// TIA Portal project "FactoryIO_Template_S7-1200_V15 (1)_V16" (V16)
// Vorlageprojekt für das Buch mit Zielsystem S7-1200

(* hardware
DEVICE "S7-1200-Station_1"  S7-1200 Station
   slot 0: "Baugruppenträger_0"  Rack  V1.0
   slot 1: "PLC_1"  CPU 1211C DC/DC/DC  6ES7 211-1AE40-0XB0  V4.1
*)

// ===== PLC "PLC_1"  CPU 1211C DC/DC/DC =====

VAR_GLOBAL   // PLC tag table "Standard-Variablentabelle"
   "visionsensor_1" AT %I0.4 : Bool;
   "pusher_1+" AT %Q0.4 : Bool;
   "pusher_1-" AT %Q0.5 : Bool;
   "pusher_2+" AT %Q0.6 : Bool;
   "visionsensor_2" AT %I0.5 : Bool;
   "visionsensor_3" AT %I0.6 : Bool;
   "visionsensor_4" AT %I0.7 : Bool;
   "pusher_2-" AT %Q0.7 : Bool;
   "pusher_3+" AT %Q1.0 : Bool;
   "pusher_3-" AT %Q1.1 : Bool;
   "pusher_4+" AT %Q1.2 : Bool;
   "pusher_4-" AT %Q1.3 : Bool;
   "Tag_1" AT %I2.5 : Bool;
   "green_moving_x" AT %I2.6 : Bool;
   "Tag_3" AT %MD10 : Time;
   "lids_sensor_bule_1" AT %I1.1 : Bool;
   "blue_lids_clamp" AT %Q2.7 : Bool;
   "blue_move_z" AT %Q2.5 : Bool;
   "blue_grab" AT %Q2.6 : Bool;
   "base_sensor_bule_1" AT %I1.2 : Bool;
   "blue_base_clamp" AT %Q3.0 : Bool;
   "bule_dectected" AT %I2.2 : Bool;
   "Tag_5" AT %MD11 : Time;
   "blue_moving_x" AT %I2.0 : Bool;
   "blue_move_x" AT %Q2.4 : Bool;
   "Tag_4" AT %MD9 : Time;
   "Tag_6" AT %MD12 : Time;
   "Tag_7" AT %MD13 : Time;
   "Start_btn" AT %I0.0 : Bool;
   "sys_on" AT %M99.0 : Bool;
   "stop_btn" AT %I0.2 : Bool;
   "emergency_stop" AT %I0.3 : Bool;
   "Tag_9" AT %M1.1 : Bool;
   "Tag_10" AT %M1.5 : Bool;
   "Tag_11" AT %M5.0 : Bool;
   "Tag_12" AT %M5.1 : Bool;
   "Tag_13" AT %M5.3 : Bool;
   "blue_base_clamped" AT %I2.4 : Bool;
   "Tag_15" AT %M6.1 : Bool;
   "blue_raise_base" AT %Q3.1 : Bool;
   "Tag_16" AT %M6.0 : Bool;
   "Tag_17" AT %M5.6 : Bool;
   "blue_base_sensor_2" AT %I1.3 : Bool;
   "Tag_18" AT %M2.6 : Bool;
   "start_light" AT %Q0.0 : Bool;
   "reset_btn" AT %I0.1 : Bool;
   "reset_light" AT %Q0.1 : Bool;
   "stop_light" AT %Q0.2 : Bool;
   "blue_lids_clamped" AT %I2.3 : Bool;
   "blue_moving_z" AT %I2.1 : Bool;
   "Tag_8" AT %M5.4 : Bool;
   "blue_lids_conveyor" AT %Q2.0 : Bool;
   "blue_base_conveyor" AT %Q2.1 : Bool;
   "Tag_19" AT %M0.7 : Bool;
   "Tag_20" AT %M0.5 : Bool;
   "Tag_21" AT %M10.1 : Bool;
   "Tag_22" AT %M11.1 : Bool;
   "Tag_23" AT %MD14 : Time;
   "Tag_24" AT %MD15 : Time;
   "green_lids_conveyor" AT %Q2.2 : Bool;
   "green_base_conveyor" AT %Q2.3 : Bool;
   "green_lids_sensor" AT %I1.4 : Bool;
   "Tag_26" AT %M1.2 : Bool;
   "green_lids_clamp" AT %Q3.5 : Bool;
   "green_base_sensor_1" AT %I1.5 : Bool;
   "Tag_25" AT %M1.6 : Bool;
   "green_base_clamp" AT %Q3.6 : Bool;
   "green_lids_clamped" AT %I3.1 : Bool;
   "green_move_z" AT %Q3.3 : Bool;
   "green_move_x" AT %Q3.2 : Bool;
   "green_detected" AT %I3.0 : Bool;
   "green_grab" AT %Q3.4 : Bool;
   "green_moving_z" AT %I2.7 : Bool;
   "Tag_27" AT %M5.5 : Bool;
   "Tag_28" AT %M5.7 : Bool;
   "Tag_2" AT %M5.2 : Bool;
   "Tag_29" AT %M6.2 : Bool;
   "Tag_30" AT %M6.3 : Bool;
   "Tag_31" AT %M6.4 : Bool;
   "green_base_raise" AT %Q3.7 : Bool;
   "green_base_sensor_2" AT %I1.6 : Bool;
   "Tag_32" AT %M2.5 : Bool;
   "Tag_33" AT %M6.5 : Bool;
   "Belt in cnc 1" AT %Q4.0 : Bool;
   "Belt in cnc 2" AT %Q4.1 : Bool;
   "Belt in cnc 3" AT %Q4.2 : Bool;
   "Belt in cnc 4" AT %Q4.3 : Bool;
   "Sensor CNC IN 1" AT %I4.0 : Bool;
   "Sensor CNC IN 2" AT %I4.1 : Bool;
   "Sensor CNC IN 3" AT %I4.2 : Bool;
   "Sensor CNC IN 4" AT %I4.3 : Bool;
   "N_SS cnc in 1" AT %M0.0 : Bool;
   "N_SS cnc in 2" AT %M0.1 : Bool;
   "N_SS cnc in 3" AT %M0.2 : Bool;
   "N_SS cnc in 4" AT %M0.3 : Bool;
   "Sensor CNC OUT 1" AT %I4.4 : Bool;
   "Sensor CNC OUT 2" AT %I4.5 : Bool;
   "Sensor CNC OUT 3" AT %I4.6 : Bool;
   "Sensor CNC OUT 4" AT %I4.7 : Bool;
   "N_SS cnc out 1" AT %M0.4 : Bool;
   "N_SS cnc out 2" AT %M0.6 : Bool;
   "N_SS cnc out 3" AT %M1.0 : Bool;
   "N_SS cnc out 4" AT %M1.3 : Bool;
   "Belt out cnc 1" AT %Q4.4 : Bool;
   "Belt out cnc 2" AT %Q4.5 : Bool;
   "Belt out cnc 3" AT %Q4.6 : Bool;
   "Belt out cnc 4" AT %Q4.7 : Bool;
   "Start CNC 1" AT %Q5.0 : Bool;
   "Start CNC 2" AT %Q5.1 : Bool;
   "Start CNC 3" AT %Q5.2 : Bool;
   "Start CNC 4" AT %Q5.3 : Bool;
   "cnc_lids_1" AT %Q6.2 : Bool;
   "cnc_lids_2" AT %Q6.3 : Bool;
   "cnc_base_1" AT %Q6.0 : Bool;
   "cnc_base_2" AT %Q6.1 : Bool;
   "Stop CNC 1" AT %Q5.4 : Bool;
   "Stop CNC 2" AT %Q5.5 : Bool;
   "Stop CNC 3" AT %Q5.6 : Bool;
   "Stop CNC 4" AT %Q5.7 : Bool;
   "conveyor_exit_cnc_1" AT %Q10.0 : Bool;
   "conveyor_exit_cnc_2" AT %Q10.1 : Bool;
   "conveyor_exit_cnc_3" AT %Q10.2 : Bool;
   "conveyor_exit_cnc_4" AT %Q10.3 : Bool;
   "conveyor_exit_cnc_5" AT %Q10.4 : Bool;
   "conveyor_exit_cnc_6" AT %Q10.5 : Bool;
   "curved_conv_assembler_in_1" AT %Q11.0 : Bool;
   "conv_assembler_in_1" AT %Q10.6 : Bool;
   "conv_assembler_in_2" AT %Q10.7 : Bool;
   "1X Set point" AT %QD44 : Real;
   "1Y Set point" AT %QD48 : Real;
   "1Z Set point" AT %QD52 : Real;
   "Roller Conveyor (4m) 2" AT %Q7.6 : Bool;
   "Roller Conveyor (6m) 1" AT %Q7.7 : Bool;
   "Belt Conveyor (6m) 8" AT %Q7.3 : Bool;
   "Belt Conveyor (6m) 13" AT %Q7.4 : Bool;
   "Roller Conveyor (4m) 3" AT %Q7.5 : Bool;
   "Pick and place (Grab)" AT %Q8.1 : Bool;
   "Retroreflective Sensor 10" AT %I7.0 : Bool;
   "Diffuse Sensor 7" AT %I6.7 : Bool;
   "Pick and place 1(Box Detected)" AT %I7.1 : Bool;
   "7M" AT %M7.0 : Bool;
   "8M" AT %M7.1 : Bool;
   "9M" AT %M7.2 : Bool;
   "12M" AT %M7.4 : Bool;
   "15M" AT %M7.7 : Bool;
   "16M" AT %M8.0 : Bool;
   "2X set point" AT %QD32 : Real;
   "2Y set point" AT %QD36 : Real;
   "2Z set point" AT %QD40 : Real;
   "Roller Conveyor 4m 1" AT %Q6.6 : Bool;
   "Roller Conveyor 6m 2" AT %Q6.7 : Bool;
   "Belt Conveyor 4m 6" AT %Q6.4 : Bool;
   "Belt Conveyor 6m 7" AT %Q6.5 : Bool;
   "Roller Conveyor 4m 4" AT %Q7.1 : Bool;
   "Pick & Place 2 Grab" AT %Q7.2 : Bool;
   "Retroreflective Sensor 11" AT %I6.4 : Bool;
   "1M" AT %M8.1 : Bool;
   "2M" AT %M8.2 : Bool;
   "Diffuse Sensor 6" AT %I6.5 : Bool;
   "3M" AT %M8.4 : Bool;
   "11M" AT %M8.7 : Bool;
   "Pick & Place 2 Box Detected" AT %I6.6 : Bool;
   "5M" AT %M8.5 : Bool;
   "6M" AT %M8.6 : Bool;
   "curved_conv_assembler_out_1" AT %Q11.1 : Bool;
   "conv_assembler_out_2" AT %Q11.2 : Bool;
   "conv_assembler_out_3" AT %Q11.3 : Bool;
   "conv_assembler_out_4" AT %Q11.4 : Bool;
   "conv_curved_in_3_axis_1" AT %Q11.5 : Bool;
   "conv_curved_in_3_axis_2" AT %Q11.6 : Bool;
   "conveyor_in_3_axis_1" AT %Q11.7 : Bool;
   "conveyor_in_3_axis_2" AT %Q12.0 : Bool;
   "conveyor_in_3_axis_3" AT %Q12.1 : Bool;
   "conveyor_in_3_axis_4" AT %Q12.2 : Bool;
   "green_base_clamped" AT %I3.2 : Bool;
END_VAR

// folder: System blocks/Program resources

DATA_BLOCK "IEC_Timer_0_DB"   // DB1
{ S7_Optimized_Access := 'TRUE' }
AUTHOR : Simatic
FAMILY : IEC
NAME : IEC_TMR
VERSION : 1.0
// stored: InstanceOfName IEC_TIMER
"IEC_TIMER"
BEGIN
END_DATA_BLOCK

DATA_BLOCK "DEM_SAN_PHAM1"   // DB2
{ S7_Optimized_Access := 'TRUE' }
AUTHOR : SIMATIC
FAMILY : IEC
NAME : DCNTR
VERSION : 1.2
// stored: InstanceOfName IEC_DCOUNTER
"IEC_DCOUNTER"
BEGIN
END_DATA_BLOCK

DATA_BLOCK "Timer0"   // DB3
{ S7_Optimized_Access := 'TRUE' }
AUTHOR : Simatic
FAMILY : IEC
NAME : IEC_TMR
VERSION : 1.0
// stored: InstanceOfName IEC_TIMER
"IEC_TIMER"
BEGIN
END_DATA_BLOCK

DATA_BLOCK "timer1"   // DB4
{ S7_Optimized_Access := 'TRUE' }
AUTHOR : Simatic
FAMILY : IEC
NAME : IEC_TMR
VERSION : 1.0
// stored: InstanceOfName IEC_TIMER
"IEC_TIMER"
BEGIN
END_DATA_BLOCK

DATA_BLOCK "DEM_SAN_PHAM"   // DB5
{ S7_Optimized_Access := 'TRUE' }
AUTHOR : Simatic
FAMILY : IEC
NAME : CNTR
VERSION : 1.0
// stored: InstanceOfName IEC_COUNTER
"IEC_COUNTER"
BEGIN
END_DATA_BLOCK

DATA_BLOCK "timer2"   // DB6
{ S7_Optimized_Access := 'TRUE' }
AUTHOR : Simatic
FAMILY : IEC
NAME : IEC_TMR
VERSION : 1.0
// stored: InstanceOfName IEC_TIMER
"IEC_TIMER"
BEGIN
END_DATA_BLOCK

DATA_BLOCK "timer4"   // DB7
{ S7_Optimized_Access := 'TRUE' }
AUTHOR : Simatic
FAMILY : IEC
NAME : IEC_TMR
VERSION : 1.0
// stored: InstanceOfName IEC_TIMER
"IEC_TIMER"
BEGIN
END_DATA_BLOCK

DATA_BLOCK "timer5"   // DB8
{ S7_Optimized_Access := 'TRUE' }
AUTHOR : Simatic
FAMILY : IEC
NAME : IEC_TMR
VERSION : 1.0
// stored: InstanceOfName IEC_TIMER
"IEC_TIMER"
BEGIN
END_DATA_BLOCK

DATA_BLOCK "timer6"   // DB9
{ S7_Optimized_Access := 'TRUE' }
AUTHOR : Simatic
FAMILY : IEC
NAME : IEC_TMR
VERSION : 1.0
// stored: InstanceOfName IEC_TIMER
"IEC_TIMER"
BEGIN
END_DATA_BLOCK

DATA_BLOCK "timer7"   // DB10
{ S7_Optimized_Access := 'TRUE' }
AUTHOR : Simatic
FAMILY : IEC
NAME : IEC_TMR
VERSION : 1.0
// stored: InstanceOfName IEC_TIMER
"IEC_TIMER"
BEGIN
END_DATA_BLOCK

DATA_BLOCK "timer8"   // DB11
{ S7_Optimized_Access := 'TRUE' }
AUTHOR : Simatic
FAMILY : IEC
NAME : IEC_TMR
VERSION : 1.0
// stored: InstanceOfName IEC_TIMER
"IEC_TIMER"
BEGIN
END_DATA_BLOCK

DATA_BLOCK "timer9"   // DB12
{ S7_Optimized_Access := 'TRUE' }
AUTHOR : Simatic
FAMILY : IEC
NAME : IEC_TMR
VERSION : 1.0
// stored: InstanceOfName IEC_TIMER
"IEC_TIMER"
BEGIN
END_DATA_BLOCK

DATA_BLOCK "timer10"   // DB13
{ S7_Optimized_Access := 'TRUE' }
AUTHOR : Simatic
FAMILY : IEC
NAME : IEC_TMR
VERSION : 1.0
// stored: InstanceOfName IEC_TIMER
"IEC_TIMER"
BEGIN
END_DATA_BLOCK

DATA_BLOCK "timer11"   // DB14
{ S7_Optimized_Access := 'TRUE' }
AUTHOR : Simatic
FAMILY : IEC
NAME : IEC_TMR
VERSION : 1.0
// stored: InstanceOfName IEC_TIMER
"IEC_TIMER"
BEGIN
END_DATA_BLOCK

DATA_BLOCK "timer12"   // DB15
{ S7_Optimized_Access := 'TRUE' }
AUTHOR : Simatic
FAMILY : IEC
NAME : IEC_TMR
VERSION : 1.0
// stored: InstanceOfName IEC_TIMER
"IEC_TIMER"
BEGIN
END_DATA_BLOCK

DATA_BLOCK "timer13"   // DB16
{ S7_Optimized_Access := 'TRUE' }
AUTHOR : Simatic
FAMILY : IEC
NAME : IEC_TMR
VERSION : 1.0
// stored: InstanceOfName IEC_TIMER
"IEC_TIMER"
BEGIN
END_DATA_BLOCK

DATA_BLOCK "timer14"   // DB17
{ S7_Optimized_Access := 'TRUE' }
AUTHOR : Simatic
FAMILY : IEC
NAME : IEC_TMR
VERSION : 1.0
// stored: InstanceOfName IEC_TIMER
"IEC_TIMER"
BEGIN
END_DATA_BLOCK

DATA_BLOCK "timer15"   // DB18
{ S7_Optimized_Access := 'TRUE' }
AUTHOR : Simatic
FAMILY : IEC
NAME : IEC_TMR
VERSION : 1.0
// stored: InstanceOfName IEC_TIMER
"IEC_TIMER"
BEGIN
END_DATA_BLOCK

DATA_BLOCK "timer16"   // DB19
{ S7_Optimized_Access := 'TRUE' }
AUTHOR : Simatic
FAMILY : IEC
NAME : IEC_TMR
VERSION : 1.0
// stored: InstanceOfName IEC_TIMER
"IEC_TIMER"
BEGIN
END_DATA_BLOCK

DATA_BLOCK "timer17"   // DB20
{ S7_Optimized_Access := 'TRUE' }
AUTHOR : Simatic
FAMILY : IEC
NAME : IEC_TMR
VERSION : 1.0
// stored: InstanceOfName IEC_TIMER
"IEC_TIMER"
BEGIN
END_DATA_BLOCK

DATA_BLOCK "timer3"   // DB21
{ S7_Optimized_Access := 'TRUE' }
AUTHOR : Simatic
FAMILY : IEC
NAME : IEC_TMR
VERSION : 1.0
// stored: InstanceOfName IEC_TIMER
"IEC_TIMER"
BEGIN
END_DATA_BLOCK

DATA_BLOCK "timer18"   // DB22
{ S7_Optimized_Access := 'TRUE' }
AUTHOR : Simatic
FAMILY : IEC
NAME : IEC_TMR
VERSION : 1.0
// stored: InstanceOfName IEC_TIMER
"IEC_TIMER"
BEGIN
END_DATA_BLOCK

DATA_BLOCK "timer19"   // DB23
{ S7_Optimized_Access := 'TRUE' }
AUTHOR : Simatic
FAMILY : IEC
NAME : IEC_TMR
VERSION : 1.0
// stored: InstanceOfName IEC_TIMER
"IEC_TIMER"
BEGIN
END_DATA_BLOCK

DATA_BLOCK "timer20"   // DB24
{ S7_Optimized_Access := 'TRUE' }
AUTHOR : Simatic
FAMILY : IEC
NAME : IEC_TMR
VERSION : 1.0
// stored: InstanceOfName IEC_TIMER
"IEC_TIMER"
BEGIN
END_DATA_BLOCK

DATA_BLOCK "timer21"   // DB25
{ S7_Optimized_Access := 'TRUE' }
AUTHOR : Simatic
FAMILY : IEC
NAME : IEC_TMR
VERSION : 1.0
// stored: InstanceOfName IEC_TIMER
"IEC_TIMER"
BEGIN
END_DATA_BLOCK

DATA_BLOCK "timer22"   // DB26
{ S7_Optimized_Access := 'TRUE' }
AUTHOR : Simatic
FAMILY : IEC
NAME : IEC_TMR
VERSION : 1.0
// stored: InstanceOfName IEC_TIMER
"IEC_TIMER"
BEGIN
END_DATA_BLOCK

DATA_BLOCK "timer23"   // DB27
{ S7_Optimized_Access := 'TRUE' }
AUTHOR : Simatic
FAMILY : IEC
NAME : IEC_TMR
VERSION : 1.0
// stored: InstanceOfName IEC_TIMER
"IEC_TIMER"
BEGIN
END_DATA_BLOCK

// folder: (top level)

FUNCTION "CNC_1" : Void   // FC1, LAD
{ S7_Optimized_Access := 'TRUE' }
VERSION : 0.1
   VAR_TEMP   // added for the SCL form of the ladder/FBD networks
      _w1 : Bool;
      _w2 : Bool;
      _w3 : Bool;
      _w4 : Bool;
   END_VAR
BEGIN

REGION Network 1: stop_cnc
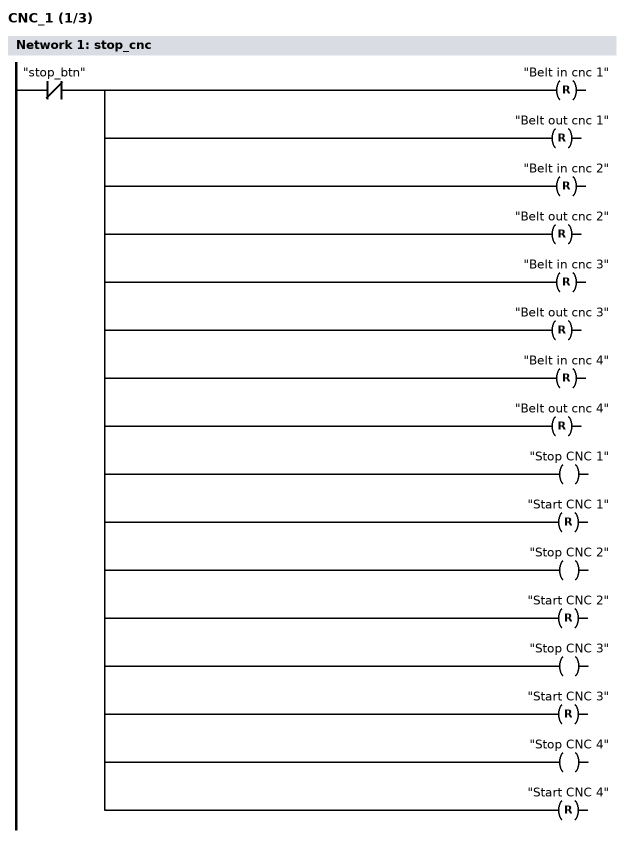
   RUNG wire#powerrail
      I_Contact( "stop_btn" )
      wire#w1
      R_Coil( "Belt in cnc 1" )
   END_RUNG
   RUNG wire#w1
      R_Coil( "Belt out cnc 1" )
   END_RUNG
   RUNG wire#w1
      R_Coil( "Belt in cnc 2" )
   END_RUNG
   RUNG wire#w1
      R_Coil( "Belt out cnc 2" )
   END_RUNG
   RUNG wire#w1
      R_Coil( "Belt in cnc 3" )
   END_RUNG
   RUNG wire#w1
      R_Coil( "Belt out cnc 3" )
   END_RUNG
   RUNG wire#w1
      R_Coil( "Belt in cnc 4" )
   END_RUNG
   RUNG wire#w1
      R_Coil( "Belt out cnc 4" )
   END_RUNG
   RUNG wire#w1
      Coil( "Stop CNC 1" )
   END_RUNG
   RUNG wire#w1
      R_Coil( "Start CNC 1" )
   END_RUNG
   RUNG wire#w1
      Coil( "Stop CNC 2" )
   END_RUNG
   RUNG wire#w1
      R_Coil( "Start CNC 2" )
   END_RUNG
   RUNG wire#w1
      Coil( "Stop CNC 3" )
   END_RUNG
   RUNG wire#w1
      R_Coil( "Start CNC 3" )
   END_RUNG
   RUNG wire#w1
      Coil( "Stop CNC 4" )
   END_RUNG
   RUNG wire#w1
      R_Coil( "Start CNC 4" )
   END_RUNG
   // the same network as SCL:
   IF NOT "stop_btn" THEN
       "Belt in cnc 1" := FALSE;
       "Belt out cnc 1" := FALSE;
       "Belt in cnc 2" := FALSE;
       "Belt out cnc 2" := FALSE;
       "Belt in cnc 3" := FALSE;
       "Belt out cnc 3" := FALSE;
       "Belt in cnc 4" := FALSE;
       "Belt out cnc 4" := FALSE;
   END_IF;
   "Stop CNC 1" := NOT "stop_btn";
   IF NOT "stop_btn" THEN "Start CNC 1" := FALSE; END_IF;
   "Stop CNC 2" := NOT "stop_btn";
   IF NOT "stop_btn" THEN "Start CNC 2" := FALSE; END_IF;
   "Stop CNC 3" := NOT "stop_btn";
   IF NOT "stop_btn" THEN "Start CNC 3" := FALSE; END_IF;
   "Stop CNC 4" := NOT "stop_btn";
   IF NOT "stop_btn" THEN "Start CNC 4" := FALSE; END_IF;
END_REGION

REGION Network 2: cnc_start
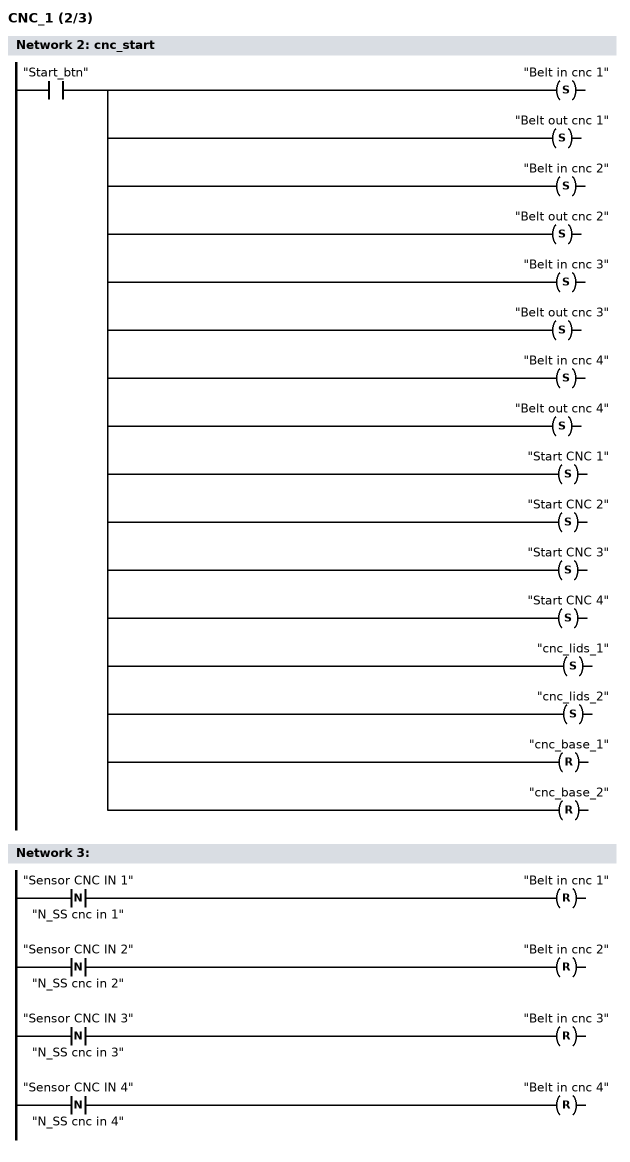
   RUNG wire#powerrail
      Contact( "Start_btn" )
      wire#w1
      S_Coil( "Belt in cnc 1" )
   END_RUNG
   RUNG wire#w1
      S_Coil( "Belt out cnc 1" )
   END_RUNG
   RUNG wire#w1
      S_Coil( "Belt in cnc 2" )
   END_RUNG
   RUNG wire#w1
      S_Coil( "Belt out cnc 2" )
   END_RUNG
   RUNG wire#w1
      S_Coil( "Belt in cnc 3" )
   END_RUNG
   RUNG wire#w1
      S_Coil( "Belt out cnc 3" )
   END_RUNG
   RUNG wire#w1
      S_Coil( "Belt in cnc 4" )
   END_RUNG
   RUNG wire#w1
      S_Coil( "Belt out cnc 4" )
   END_RUNG
   RUNG wire#w1
      S_Coil( "Start CNC 1" )
   END_RUNG
   RUNG wire#w1
      S_Coil( "Start CNC 2" )
   END_RUNG
   RUNG wire#w1
      S_Coil( "Start CNC 3" )
   END_RUNG
   RUNG wire#w1
      S_Coil( "Start CNC 4" )
   END_RUNG
   RUNG wire#w1
      S_Coil( "cnc_lids_1" )
   END_RUNG
   RUNG wire#w1
      S_Coil( "cnc_lids_2" )
   END_RUNG
   RUNG wire#w1
      R_Coil( "cnc_base_1" )
   END_RUNG
   RUNG wire#w1
      R_Coil( "cnc_base_2" )
   END_RUNG
   // the same network as SCL:
   IF "Start_btn" THEN
       "Belt in cnc 1" := TRUE;
       "Belt out cnc 1" := TRUE;
       "Belt in cnc 2" := TRUE;
       "Belt out cnc 2" := TRUE;
       "Belt in cnc 3" := TRUE;
       "Belt out cnc 3" := TRUE;
       "Belt in cnc 4" := TRUE;
       "Belt out cnc 4" := TRUE;
       "Start CNC 1" := TRUE;
       "Start CNC 2" := TRUE;
       "Start CNC 3" := TRUE;
       "Start CNC 4" := TRUE;
       "cnc_lids_1" := TRUE;
       "cnc_lids_2" := TRUE;
       "cnc_base_1" := FALSE;
       "cnc_base_2" := FALSE;
   END_IF;
END_REGION

REGION Network 3
   RUNG wire#powerrail
      N_Contact(operand := "Sensor CNC IN 1", bit := "N_SS cnc in 1")
      R_Coil( "Belt in cnc 1" )
   END_RUNG
   RUNG wire#powerrail
      N_Contact(operand := "Sensor CNC IN 2", bit := "N_SS cnc in 2")
      R_Coil( "Belt in cnc 2" )
   END_RUNG
   RUNG wire#powerrail
      N_Contact(operand := "Sensor CNC IN 3", bit := "N_SS cnc in 3")
      R_Coil( "Belt in cnc 3" )
   END_RUNG
   RUNG wire#powerrail
      N_Contact(operand := "Sensor CNC IN 4", bit := "N_SS cnc in 4")
      R_Coil( "Belt in cnc 4" )
   END_RUNG
   // the same network as SCL:
   #_w1 := NOT "Sensor CNC IN 1" AND "N_SS cnc in 1";   // falling edge of "Sensor CNC IN 1"
   "N_SS cnc in 1" := "Sensor CNC IN 1";
   IF #_w1 THEN "Belt in cnc 1" := FALSE; END_IF;
   #_w2 := NOT "Sensor CNC IN 2" AND "N_SS cnc in 2";   // falling edge of "Sensor CNC IN 2"
   "N_SS cnc in 2" := "Sensor CNC IN 2";
   IF #_w2 THEN "Belt in cnc 2" := FALSE; END_IF;
   #_w3 := NOT "Sensor CNC IN 3" AND "N_SS cnc in 3";   // falling edge of "Sensor CNC IN 3"
   "N_SS cnc in 3" := "Sensor CNC IN 3";
   IF #_w3 THEN "Belt in cnc 3" := FALSE; END_IF;
   #_w4 := NOT "Sensor CNC IN 4" AND "N_SS cnc in 4";   // falling edge of "Sensor CNC IN 4"
   "N_SS cnc in 4" := "Sensor CNC IN 4";
   IF #_w4 THEN "Belt in cnc 4" := FALSE; END_IF;
END_REGION

REGION Network 4: as
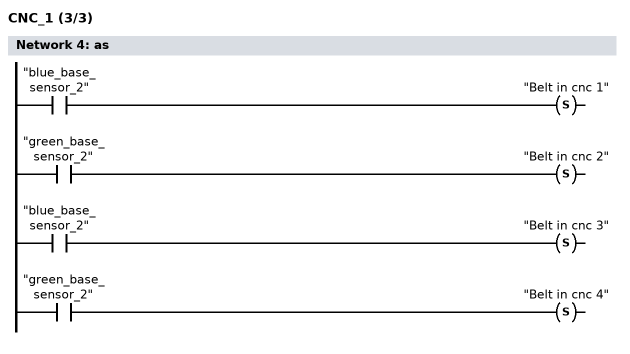
   RUNG wire#powerrail
      Contact( "blue_base_sensor_2" )
      S_Coil( "Belt in cnc 1" )
   END_RUNG
   RUNG wire#powerrail
      Contact( "green_base_sensor_2" )
      S_Coil( "Belt in cnc 2" )
   END_RUNG
   RUNG wire#powerrail
      Contact( "blue_base_sensor_2" )
      S_Coil( "Belt in cnc 3" )
   END_RUNG
   RUNG wire#powerrail
      Contact( "green_base_sensor_2" )
      S_Coil( "Belt in cnc 4" )
   END_RUNG
   // the same network as SCL:
   IF "blue_base_sensor_2" THEN "Belt in cnc 1" := TRUE; END_IF;
   IF "green_base_sensor_2" THEN "Belt in cnc 2" := TRUE; END_IF;
   IF "blue_base_sensor_2" THEN "Belt in cnc 3" := TRUE; END_IF;
   IF "green_base_sensor_2" THEN "Belt in cnc 4" := TRUE; END_IF;
END_REGION
END_FUNCTION

FUNCTION "pusher" : Void   // FC2, LAD
{ S7_Optimized_Access := 'TRUE' }
VERSION : 0.1
BEGIN

REGION Network 1
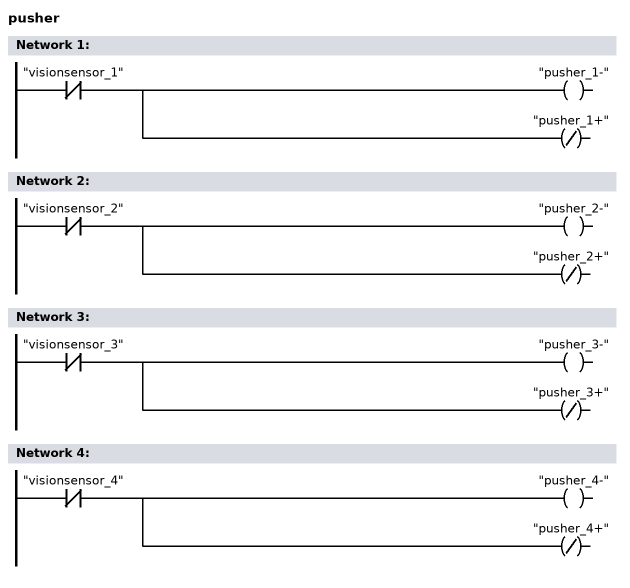
   RUNG wire#powerrail
      I_Contact( "visionsensor_1" )
      wire#w1
      Coil( "pusher_1-" )
   END_RUNG
   RUNG wire#w1
      I_Coil( "pusher_1+" )
   END_RUNG
   // the same network as SCL:
   "pusher_1-" := NOT "visionsensor_1";
   "pusher_1+" := NOT (NOT "visionsensor_1");
END_REGION

REGION Network 2
   RUNG wire#powerrail
      I_Contact( "visionsensor_2" )
      wire#w1
      Coil( "pusher_2-" )
   END_RUNG
   RUNG wire#w1
      I_Coil( "pusher_2+" )
   END_RUNG
   // the same network as SCL:
   "pusher_2-" := NOT "visionsensor_2";
   "pusher_2+" := NOT (NOT "visionsensor_2");
END_REGION

REGION Network 3
   RUNG wire#powerrail
      I_Contact( "visionsensor_3" )
      wire#w1
      Coil( "pusher_3-" )
   END_RUNG
   RUNG wire#w1
      I_Coil( "pusher_3+" )
   END_RUNG
   // the same network as SCL:
   "pusher_3-" := NOT "visionsensor_3";
   "pusher_3+" := NOT (NOT "visionsensor_3");
END_REGION

REGION Network 4
   RUNG wire#powerrail
      I_Contact( "visionsensor_4" )
      wire#w1
      Coil( "pusher_4-" )
   END_RUNG
   RUNG wire#w1
      I_Coil( "pusher_4+" )
   END_RUNG
   // the same network as SCL:
   "pusher_4-" := NOT "visionsensor_4";
   "pusher_4+" := NOT (NOT "visionsensor_4");
END_REGION
END_FUNCTION

FUNCTION "control_conveyor" : Void   // FC3, LAD
{ S7_Optimized_Access := 'TRUE' }
VERSION : 0.1
BEGIN

REGION Network 1: start conveyor
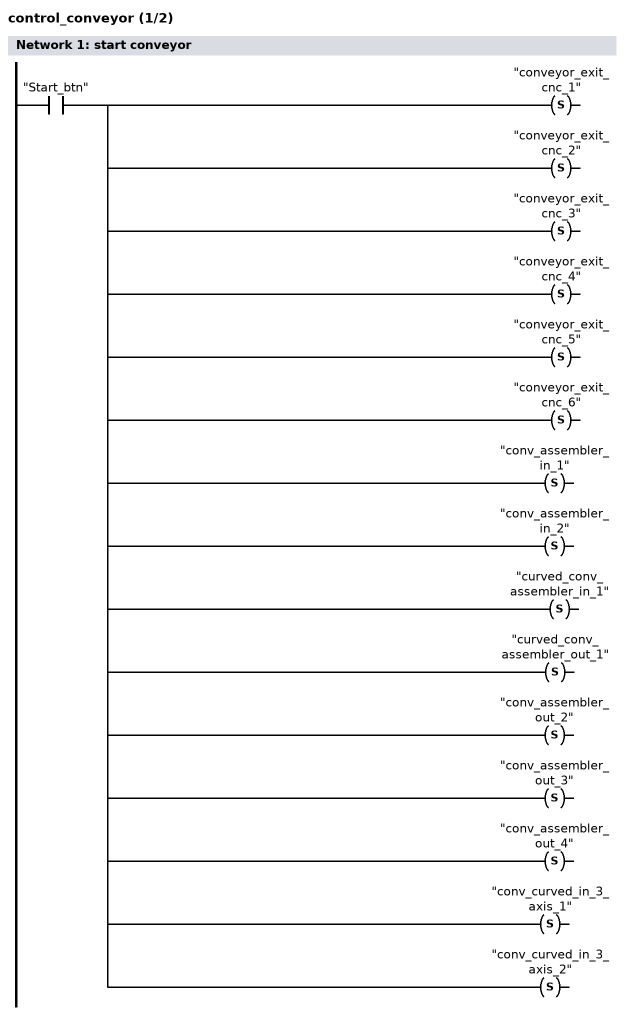
   RUNG wire#powerrail
      Contact( "Start_btn" )
      wire#w1
      S_Coil( "conveyor_exit_cnc_1" )
   END_RUNG
   RUNG wire#w1
      S_Coil( "conveyor_exit_cnc_2" )
   END_RUNG
   RUNG wire#w1
      S_Coil( "conveyor_exit_cnc_3" )
   END_RUNG
   RUNG wire#w1
      S_Coil( "conveyor_exit_cnc_4" )
   END_RUNG
   RUNG wire#w1
      S_Coil( "conveyor_exit_cnc_5" )
   END_RUNG
   RUNG wire#w1
      S_Coil( "conveyor_exit_cnc_6" )
   END_RUNG
   RUNG wire#w1
      S_Coil( "conv_assembler_in_1" )
   END_RUNG
   RUNG wire#w1
      S_Coil( "conv_assembler_in_2" )
   END_RUNG
   RUNG wire#w1
      S_Coil( "curved_conv_assembler_in_1" )
   END_RUNG
   RUNG wire#w1
      S_Coil( "curved_conv_assembler_out_1" )
   END_RUNG
   RUNG wire#w1
      S_Coil( "conv_assembler_out_2" )
   END_RUNG
   RUNG wire#w1
      S_Coil( "conv_assembler_out_3" )
   END_RUNG
   RUNG wire#w1
      S_Coil( "conv_assembler_out_4" )
   END_RUNG
   RUNG wire#w1
      S_Coil( "conv_curved_in_3_axis_1" )
   END_RUNG
   RUNG wire#w1
      S_Coil( "conv_curved_in_3_axis_2" )
   END_RUNG
   // the same network as SCL:
   IF "Start_btn" THEN
       "conveyor_exit_cnc_1" := TRUE;
       "conveyor_exit_cnc_2" := TRUE;
       "conveyor_exit_cnc_3" := TRUE;
       "conveyor_exit_cnc_4" := TRUE;
       "conveyor_exit_cnc_5" := TRUE;
       "conveyor_exit_cnc_6" := TRUE;
       "conv_assembler_in_1" := TRUE;
       "conv_assembler_in_2" := TRUE;
       "curved_conv_assembler_in_1" := TRUE;
       "curved_conv_assembler_out_1" := TRUE;
       "conv_assembler_out_2" := TRUE;
       "conv_assembler_out_3" := TRUE;
       "conv_assembler_out_4" := TRUE;
       "conv_curved_in_3_axis_1" := TRUE;
       "conv_curved_in_3_axis_2" := TRUE;
   END_IF;
END_REGION

REGION Network 2: start conveyor
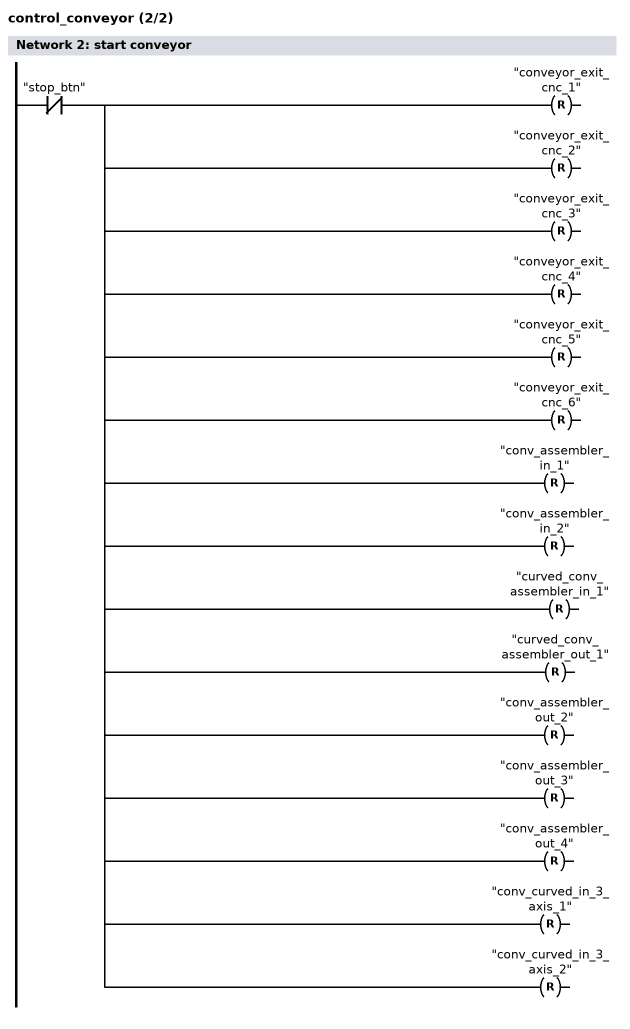
   RUNG wire#powerrail
      I_Contact( "stop_btn" )
      wire#w1
      R_Coil( "conveyor_exit_cnc_1" )
   END_RUNG
   RUNG wire#w1
      R_Coil( "conveyor_exit_cnc_2" )
   END_RUNG
   RUNG wire#w1
      R_Coil( "conveyor_exit_cnc_3" )
   END_RUNG
   RUNG wire#w1
      R_Coil( "conveyor_exit_cnc_4" )
   END_RUNG
   RUNG wire#w1
      R_Coil( "conveyor_exit_cnc_5" )
   END_RUNG
   RUNG wire#w1
      R_Coil( "conveyor_exit_cnc_6" )
   END_RUNG
   RUNG wire#w1
      R_Coil( "conv_assembler_in_1" )
   END_RUNG
   RUNG wire#w1
      R_Coil( "conv_assembler_in_2" )
   END_RUNG
   RUNG wire#w1
      R_Coil( "curved_conv_assembler_in_1" )
   END_RUNG
   RUNG wire#w1
      R_Coil( "curved_conv_assembler_out_1" )
   END_RUNG
   RUNG wire#w1
      R_Coil( "conv_assembler_out_2" )
   END_RUNG
   RUNG wire#w1
      R_Coil( "conv_assembler_out_3" )
   END_RUNG
   RUNG wire#w1
      R_Coil( "conv_assembler_out_4" )
   END_RUNG
   RUNG wire#w1
      R_Coil( "conv_curved_in_3_axis_1" )
   END_RUNG
   RUNG wire#w1
      R_Coil( "conv_curved_in_3_axis_2" )
   END_RUNG
   // the same network as SCL:
   IF NOT "stop_btn" THEN
       "conveyor_exit_cnc_1" := FALSE;
       "conveyor_exit_cnc_2" := FALSE;
       "conveyor_exit_cnc_3" := FALSE;
       "conveyor_exit_cnc_4" := FALSE;
       "conveyor_exit_cnc_5" := FALSE;
       "conveyor_exit_cnc_6" := FALSE;
       "conv_assembler_in_1" := FALSE;
       "conv_assembler_in_2" := FALSE;
       "curved_conv_assembler_in_1" := FALSE;
       "curved_conv_assembler_out_1" := FALSE;
       "conv_assembler_out_2" := FALSE;
       "conv_assembler_out_3" := FALSE;
       "conv_assembler_out_4" := FALSE;
       "conv_curved_in_3_axis_1" := FALSE;
       "conv_curved_in_3_axis_2" := FALSE;
   END_IF;
END_REGION
END_FUNCTION

FUNCTION "two axis" : Void   // FC4, LAD
{ S7_Optimized_Access := 'TRUE' }
VERSION : 0.1
   VAR_TEMP   // added for the SCL form of the ladder/FBD networks
      _w1 : Bool;
      _w2 : Bool;
   END_VAR
BEGIN

REGION Network 1: start stop
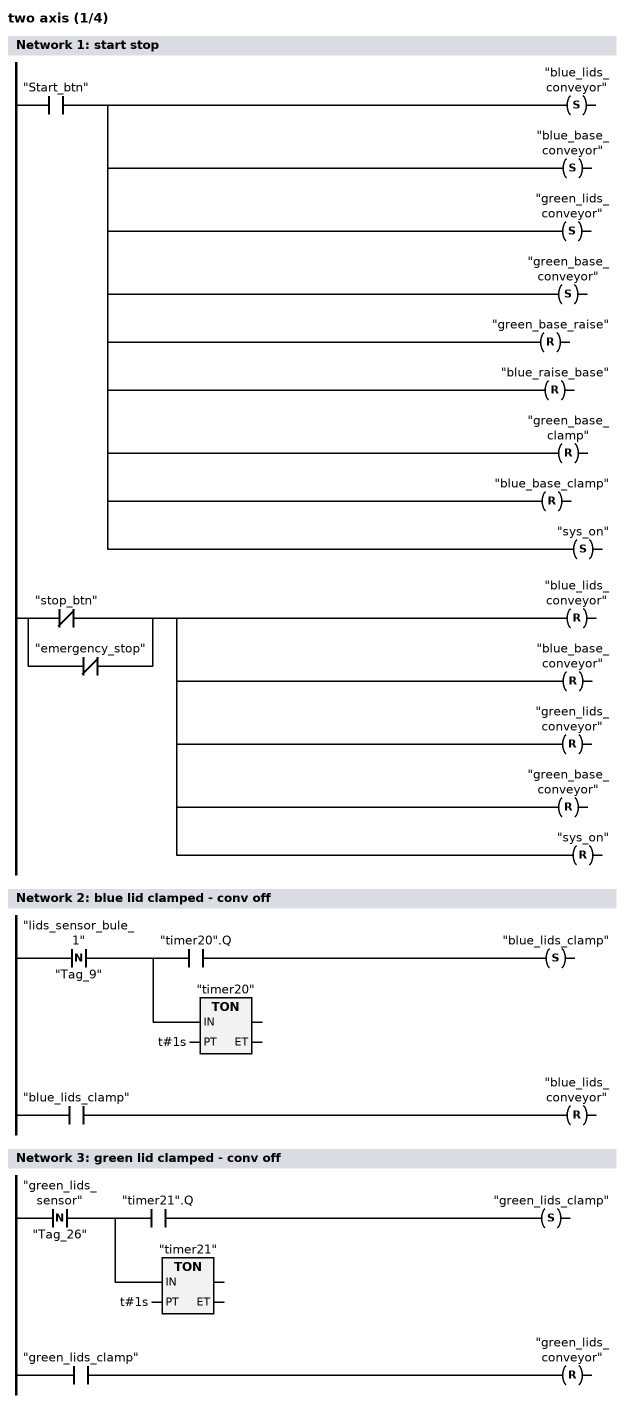
   RUNG wire#powerrail
      Contact( "Start_btn" )
      wire#w1
      S_Coil( "blue_lids_conveyor" )
   END_RUNG
   RUNG wire#w1
      S_Coil( "blue_base_conveyor" )
   END_RUNG
   RUNG wire#w1
      S_Coil( "green_lids_conveyor" )
   END_RUNG
   RUNG wire#w1
      S_Coil( "green_base_conveyor" )
   END_RUNG
   RUNG wire#w1
      R_Coil( "green_base_raise" )
   END_RUNG
   RUNG wire#w1
      R_Coil( "blue_raise_base" )
   END_RUNG
   RUNG wire#w1
      R_Coil( "green_base_clamp" )
   END_RUNG
   RUNG wire#w1
      R_Coil( "blue_base_clamp" )
   END_RUNG
   RUNG wire#w1
      S_Coil( "sys_on" )
   END_RUNG
   RUNG wire#powerrail
      I_Contact( "stop_btn" )
      wire#w2
      R_Coil( "blue_lids_conveyor" )
   END_RUNG
   RUNG wire#powerrail
      I_Contact( "emergency_stop" )
   END_RUNG wire#w2
   RUNG wire#w2
      R_Coil( "blue_base_conveyor" )
   END_RUNG
   RUNG wire#w2
      R_Coil( "green_lids_conveyor" )
   END_RUNG
   RUNG wire#w2
      R_Coil( "green_base_conveyor" )
   END_RUNG
   RUNG wire#w2
      R_Coil( "sys_on" )
   END_RUNG
   // the same network as SCL:
   IF "Start_btn" THEN
       "blue_lids_conveyor" := TRUE;
       "blue_base_conveyor" := TRUE;
       "green_lids_conveyor" := TRUE;
       "green_base_conveyor" := TRUE;
       "green_base_raise" := FALSE;
       "blue_raise_base" := FALSE;
       "green_base_clamp" := FALSE;
       "blue_base_clamp" := FALSE;
       "sys_on" := TRUE;
   END_IF;
   IF NOT "stop_btn" OR NOT "emergency_stop" THEN
       "blue_lids_conveyor" := FALSE;
       "blue_base_conveyor" := FALSE;
       "green_lids_conveyor" := FALSE;
       "green_base_conveyor" := FALSE;
       "sys_on" := FALSE;
   END_IF;
END_REGION

REGION Network 2: blue lid clamped - conv off
   #_w1 := NOT "lids_sensor_bule_1" AND "Tag_9";   // falling edge of "lids_sensor_bule_1"
   "Tag_9" := "lids_sensor_bule_1";
   IF #_w1 AND "timer20".Q THEN "blue_lids_clamp" := TRUE; END_IF;
   "timer20".TON(IN := #_w1, PT := t#1s);
   IF "blue_lids_clamp" THEN "blue_lids_conveyor" := FALSE; END_IF;
END_REGION

REGION Network 3: green lid clamped - conv off
   #_w1 := NOT "green_lids_sensor" AND "Tag_26";   // falling edge of "green_lids_sensor"
   "Tag_26" := "green_lids_sensor";
   IF #_w1 AND "timer21".Q THEN "green_lids_clamp" := TRUE; END_IF;
   "timer21".TON(IN := #_w1, PT := t#1s);
   IF "green_lids_clamp" THEN "green_lids_conveyor" := FALSE; END_IF;
END_REGION

REGION Network 4: blue base clamped - conv off
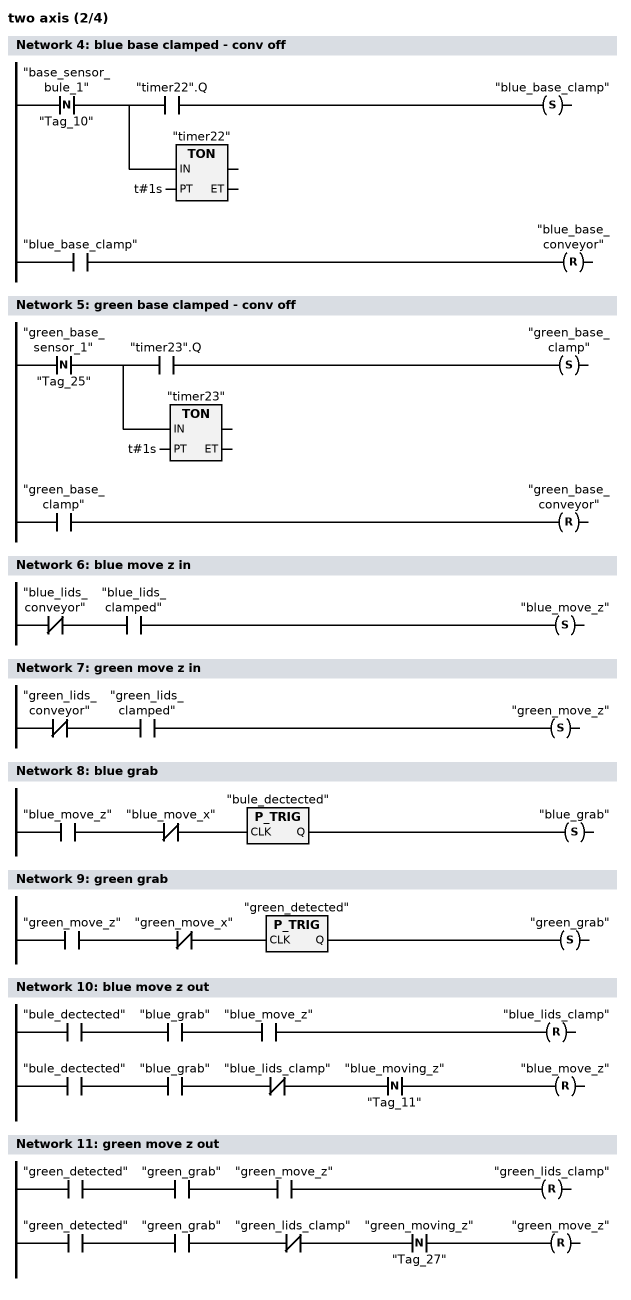
   #_w1 := NOT "base_sensor_bule_1" AND "Tag_10";   // falling edge of "base_sensor_bule_1"
   "Tag_10" := "base_sensor_bule_1";
   IF #_w1 AND "timer22".Q THEN "blue_base_clamp" := TRUE; END_IF;
   "timer22".TON(IN := #_w1, PT := t#1s);
   IF "blue_base_clamp" THEN "blue_base_conveyor" := FALSE; END_IF;
END_REGION

REGION Network 5: green base clamped - conv off
   #_w1 := NOT "green_base_sensor_1" AND "Tag_25";   // falling edge of "green_base_sensor_1"
   "Tag_25" := "green_base_sensor_1";
   IF #_w1 AND "timer23".Q THEN "green_base_clamp" := TRUE; END_IF;
   "timer23".TON(IN := #_w1, PT := t#1s);
   IF "green_base_clamp" THEN "green_base_conveyor" := FALSE; END_IF;
END_REGION

REGION Network 6: blue move z in
   RUNG wire#powerrail
      I_Contact( "blue_lids_conveyor" )
      Contact( "blue_lids_clamped" )
      S_Coil( "blue_move_z" )
   END_RUNG
   // the same network as SCL:
   IF NOT "blue_lids_conveyor" AND "blue_lids_clamped" THEN "blue_move_z" := TRUE; END_IF;
END_REGION

REGION Network 7: green move z in
   RUNG wire#powerrail
      I_Contact( "green_lids_conveyor" )
      Contact( "green_lids_clamped" )
      S_Coil( "green_move_z" )
   END_RUNG
   // the same network as SCL:
   IF NOT "green_lids_conveyor" AND "green_lids_clamped" THEN "green_move_z" := TRUE; END_IF;
END_REGION

REGION Network 8: blue grab
   RUNG wire#powerrail
      Contact( "blue_move_z" )
      I_Contact( "blue_move_x" )
      P_Trig( "bule_dectected" )
      S_Coil( "blue_grab" )
   END_RUNG
   // the same network as SCL:
   #_w1 := "blue_move_z" AND NOT "blue_move_x";
   #_w2 := #_w1 AND NOT "bule_dectected";   // rising edge
   "bule_dectected" := #_w1;
   IF #_w2 THEN "blue_grab" := TRUE; END_IF;
END_REGION

REGION Network 9: green grab
   RUNG wire#powerrail
      Contact( "green_move_z" )
      I_Contact( "green_move_x" )
      P_Trig( "green_detected" )
      S_Coil( "green_grab" )
   END_RUNG
   // the same network as SCL:
   #_w1 := "green_move_z" AND NOT "green_move_x";
   #_w2 := #_w1 AND NOT "green_detected";   // rising edge
   "green_detected" := #_w1;
   IF #_w2 THEN "green_grab" := TRUE; END_IF;
END_REGION

REGION Network 10: blue move z out
   RUNG wire#powerrail
      Contact( "bule_dectected" )
      Contact( "blue_grab" )
      Contact( "blue_move_z" )
      R_Coil( "blue_lids_clamp" )
   END_RUNG
   RUNG wire#powerrail
      Contact( "bule_dectected" )
      Contact( "blue_grab" )
      I_Contact( "blue_lids_clamp" )
      N_Contact(operand := "blue_moving_z", bit := "Tag_11")
      R_Coil( "blue_move_z" )
   END_RUNG
   // the same network as SCL:
   IF "bule_dectected" AND "blue_grab" AND "blue_move_z" THEN "blue_lids_clamp" := FALSE; END_IF;
   #_w1 := "bule_dectected" AND "blue_grab" AND NOT "blue_lids_clamp" AND NOT "blue_moving_z" AND "Tag_11";   // falling edge of "blue_moving_z"
   "Tag_11" := "blue_moving_z";
   IF #_w1 THEN "blue_move_z" := FALSE; END_IF;
END_REGION

REGION Network 11: green move z out
   RUNG wire#powerrail
      Contact( "green_detected" )
      Contact( "green_grab" )
      Contact( "green_move_z" )
      R_Coil( "green_lids_clamp" )
   END_RUNG
   RUNG wire#powerrail
      Contact( "green_detected" )
      Contact( "green_grab" )
      I_Contact( "green_lids_clamp" )
      N_Contact(operand := "green_moving_z", bit := "Tag_27")
      R_Coil( "green_move_z" )
   END_RUNG
   // the same network as SCL:
   IF "green_detected" AND "green_grab" AND "green_move_z" THEN "green_lids_clamp" := FALSE; END_IF;
   #_w1 := "green_detected" AND "green_grab" AND NOT "green_lids_clamp" AND NOT "green_moving_z" AND "Tag_27";   // falling edge of "green_moving_z"
   "Tag_27" := "green_moving_z";
   IF #_w1 THEN "green_move_z" := FALSE; END_IF;
END_REGION

REGION Network 12: blue move x
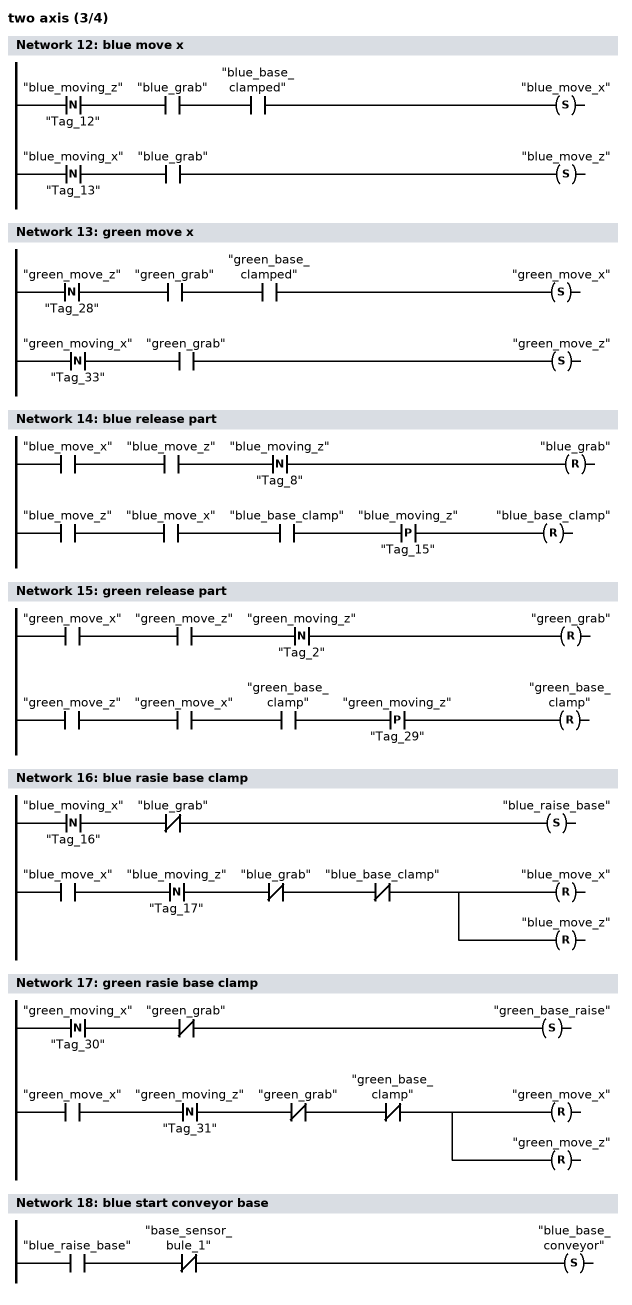
   RUNG wire#powerrail
      N_Contact(operand := "blue_moving_z", bit := "Tag_12")
      Contact( "blue_grab" )
      Contact( "blue_base_clamped" )
      S_Coil( "blue_move_x" )
   END_RUNG
   RUNG wire#powerrail
      N_Contact(operand := "blue_moving_x", bit := "Tag_13")
      Contact( "blue_grab" )
      S_Coil( "blue_move_z" )
   END_RUNG
   // the same network as SCL:
   #_w1 := NOT "blue_moving_z" AND "Tag_12";   // falling edge of "blue_moving_z"
   "Tag_12" := "blue_moving_z";
   IF #_w1 AND "blue_grab" AND "blue_base_clamped" THEN "blue_move_x" := TRUE; END_IF;
   #_w2 := NOT "blue_moving_x" AND "Tag_13";   // falling edge of "blue_moving_x"
   "Tag_13" := "blue_moving_x";
   IF #_w2 AND "blue_grab" THEN "blue_move_z" := TRUE; END_IF;
END_REGION

REGION Network 13: green move x
   RUNG wire#powerrail
      N_Contact(operand := "green_move_z", bit := "Tag_28")
      Contact( "green_grab" )
      Contact( "green_base_clamped" )
      S_Coil( "green_move_x" )
   END_RUNG
   RUNG wire#powerrail
      N_Contact(operand := "green_moving_x", bit := "Tag_33")
      Contact( "green_grab" )
      S_Coil( "green_move_z" )
   END_RUNG
   // the same network as SCL:
   #_w1 := NOT "green_move_z" AND "Tag_28";   // falling edge of "green_move_z"
   "Tag_28" := "green_move_z";
   IF #_w1 AND "green_grab" AND "green_base_clamped" THEN "green_move_x" := TRUE; END_IF;
   #_w2 := NOT "green_moving_x" AND "Tag_33";   // falling edge of "green_moving_x"
   "Tag_33" := "green_moving_x";
   IF #_w2 AND "green_grab" THEN "green_move_z" := TRUE; END_IF;
END_REGION

REGION Network 14: blue release part
   RUNG wire#powerrail
      Contact( "blue_move_x" )
      Contact( "blue_move_z" )
      N_Contact(operand := "blue_moving_z", bit := "Tag_8")
      R_Coil( "blue_grab" )
   END_RUNG
   RUNG wire#powerrail
      Contact( "blue_move_z" )
      Contact( "blue_move_x" )
      Contact( "blue_base_clamp" )
      P_Contact(operand := "blue_moving_z", bit := "Tag_15")
      R_Coil( "blue_base_clamp" )
   END_RUNG
   // the same network as SCL:
   #_w1 := "blue_move_x" AND "blue_move_z" AND NOT "blue_moving_z" AND "Tag_8";   // falling edge of "blue_moving_z"
   "Tag_8" := "blue_moving_z";
   IF #_w1 THEN "blue_grab" := FALSE; END_IF;
   #_w2 := "blue_move_z" AND "blue_move_x" AND "blue_base_clamp" AND "blue_moving_z" AND NOT "Tag_15";   // rising edge of "blue_moving_z"
   "Tag_15" := "blue_moving_z";
   IF #_w2 THEN "blue_base_clamp" := FALSE; END_IF;
END_REGION

REGION Network 15: green release part
   RUNG wire#powerrail
      Contact( "green_move_x" )
      Contact( "green_move_z" )
      N_Contact(operand := "green_moving_z", bit := "Tag_2")
      R_Coil( "green_grab" )
   END_RUNG
   RUNG wire#powerrail
      Contact( "green_move_z" )
      Contact( "green_move_x" )
      Contact( "green_base_clamp" )
      P_Contact(operand := "green_moving_z", bit := "Tag_29")
      R_Coil( "green_base_clamp" )
   END_RUNG
   // the same network as SCL:
   #_w1 := "green_move_x" AND "green_move_z" AND NOT "green_moving_z" AND "Tag_2";   // falling edge of "green_moving_z"
   "Tag_2" := "green_moving_z";
   IF #_w1 THEN "green_grab" := FALSE; END_IF;
   #_w2 := "green_move_z" AND "green_move_x" AND "green_base_clamp" AND "green_moving_z" AND NOT "Tag_29";   // rising edge of "green_moving_z"
   "Tag_29" := "green_moving_z";
   IF #_w2 THEN "green_base_clamp" := FALSE; END_IF;
END_REGION

REGION Network 16: blue rasie base clamp
   RUNG wire#powerrail
      N_Contact(operand := "blue_moving_x", bit := "Tag_16")
      I_Contact( "blue_grab" )
      S_Coil( "blue_raise_base" )
   END_RUNG
   RUNG wire#powerrail
      Contact( "blue_move_x" )
      N_Contact(operand := "blue_moving_z", bit := "Tag_17")
      I_Contact( "blue_grab" )
      I_Contact( "blue_base_clamp" )
      wire#w1
      R_Coil( "blue_move_x" )
   END_RUNG
   RUNG wire#w1
      R_Coil( "blue_move_z" )
   END_RUNG
   // the same network as SCL:
   #_w1 := NOT "blue_moving_x" AND "Tag_16";   // falling edge of "blue_moving_x"
   "Tag_16" := "blue_moving_x";
   IF #_w1 AND NOT "blue_grab" THEN "blue_raise_base" := TRUE; END_IF;
   #_w2 := "blue_move_x" AND NOT "blue_moving_z" AND "Tag_17";   // falling edge of "blue_moving_z"
   "Tag_17" := "blue_moving_z";
   IF #_w2 AND NOT "blue_grab" AND NOT "blue_base_clamp" THEN
       "blue_move_x" := FALSE;
       "blue_move_z" := FALSE;
   END_IF;
END_REGION

REGION Network 17: green rasie base clamp
   RUNG wire#powerrail
      N_Contact(operand := "green_moving_x", bit := "Tag_30")
      I_Contact( "green_grab" )
      S_Coil( "green_base_raise" )
   END_RUNG
   RUNG wire#powerrail
      Contact( "green_move_x" )
      N_Contact(operand := "green_moving_z", bit := "Tag_31")
      I_Contact( "green_grab" )
      I_Contact( "green_base_clamp" )
      wire#w1
      R_Coil( "green_move_x" )
   END_RUNG
   RUNG wire#w1
      R_Coil( "green_move_z" )
   END_RUNG
   // the same network as SCL:
   #_w1 := NOT "green_moving_x" AND "Tag_30";   // falling edge of "green_moving_x"
   "Tag_30" := "green_moving_x";
   IF #_w1 AND NOT "green_grab" THEN "green_base_raise" := TRUE; END_IF;
   #_w2 := "green_move_x" AND NOT "green_moving_z" AND "Tag_31";   // falling edge of "green_moving_z"
   "Tag_31" := "green_moving_z";
   IF #_w2 AND NOT "green_grab" AND NOT "green_base_clamp" THEN
       "green_move_x" := FALSE;
       "green_move_z" := FALSE;
   END_IF;
END_REGION

REGION Network 18: blue start conveyor base
   RUNG wire#powerrail
      Contact( "blue_raise_base" )
      I_Contact( "base_sensor_bule_1" )
      S_Coil( "blue_base_conveyor" )
   END_RUNG
   // the same network as SCL:
   IF "blue_raise_base" AND NOT "base_sensor_bule_1" THEN "blue_base_conveyor" := TRUE; END_IF;
END_REGION

REGION Network 19: green start conveyor base
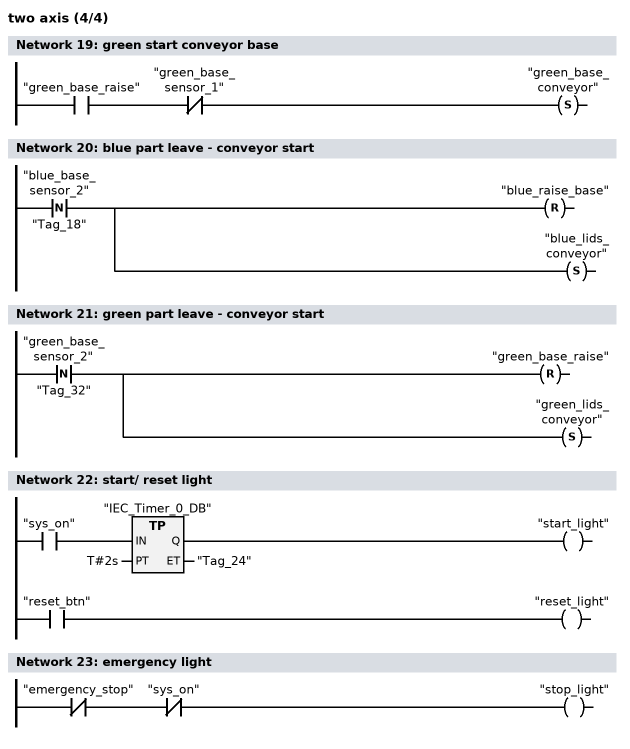
   RUNG wire#powerrail
      Contact( "green_base_raise" )
      I_Contact( "green_base_sensor_1" )
      S_Coil( "green_base_conveyor" )
   END_RUNG
   // the same network as SCL:
   IF "green_base_raise" AND NOT "green_base_sensor_1" THEN "green_base_conveyor" := TRUE; END_IF;
END_REGION

REGION Network 20: blue part leave - conveyor start
   RUNG wire#powerrail
      N_Contact(operand := "blue_base_sensor_2", bit := "Tag_18")
      wire#w1
      R_Coil( "blue_raise_base" )
   END_RUNG
   RUNG wire#w1
      S_Coil( "blue_lids_conveyor" )
   END_RUNG
   // the same network as SCL:
   #_w1 := NOT "blue_base_sensor_2" AND "Tag_18";   // falling edge of "blue_base_sensor_2"
   "Tag_18" := "blue_base_sensor_2";
   IF #_w1 THEN
       "blue_raise_base" := FALSE;
       "blue_lids_conveyor" := TRUE;
   END_IF;
END_REGION

REGION Network 21: green part leave - conveyor start
   RUNG wire#powerrail
      N_Contact(operand := "green_base_sensor_2", bit := "Tag_32")
      wire#w1
      R_Coil( "green_base_raise" )
   END_RUNG
   RUNG wire#w1
      S_Coil( "green_lids_conveyor" )
   END_RUNG
   // the same network as SCL:
   #_w1 := NOT "green_base_sensor_2" AND "Tag_32";   // falling edge of "green_base_sensor_2"
   "Tag_32" := "green_base_sensor_2";
   IF #_w1 THEN
       "green_base_raise" := FALSE;
       "green_lids_conveyor" := TRUE;
   END_IF;
END_REGION

REGION Network 22: start/ reset light
   "IEC_Timer_0_DB".TP(IN := "sys_on", PT := T#2s, ET => "Tag_24");
   "start_light" := "IEC_Timer_0_DB".Q;
   "reset_light" := "reset_btn";
END_REGION

REGION Network 23: emergency light
   RUNG wire#powerrail
      I_Contact( "emergency_stop" )
      I_Contact( "sys_on" )
      Coil( "stop_light" )
   END_RUNG
   // the same network as SCL:
   "stop_light" := NOT "emergency_stop" AND NOT "sys_on";
END_REGION
END_FUNCTION

FUNCTION "PICK_AND_PLACE1" : Void   // FC5, LAD
{ S7_Optimized_Access := 'TRUE' }
VERSION : 0.1
   VAR_TEMP   // added for the SCL form of the ladder/FBD networks
      _w1 : Bool;
      _w2 : Bool;
      _w3 : Bool;
   END_VAR
BEGIN

REGION Network 1
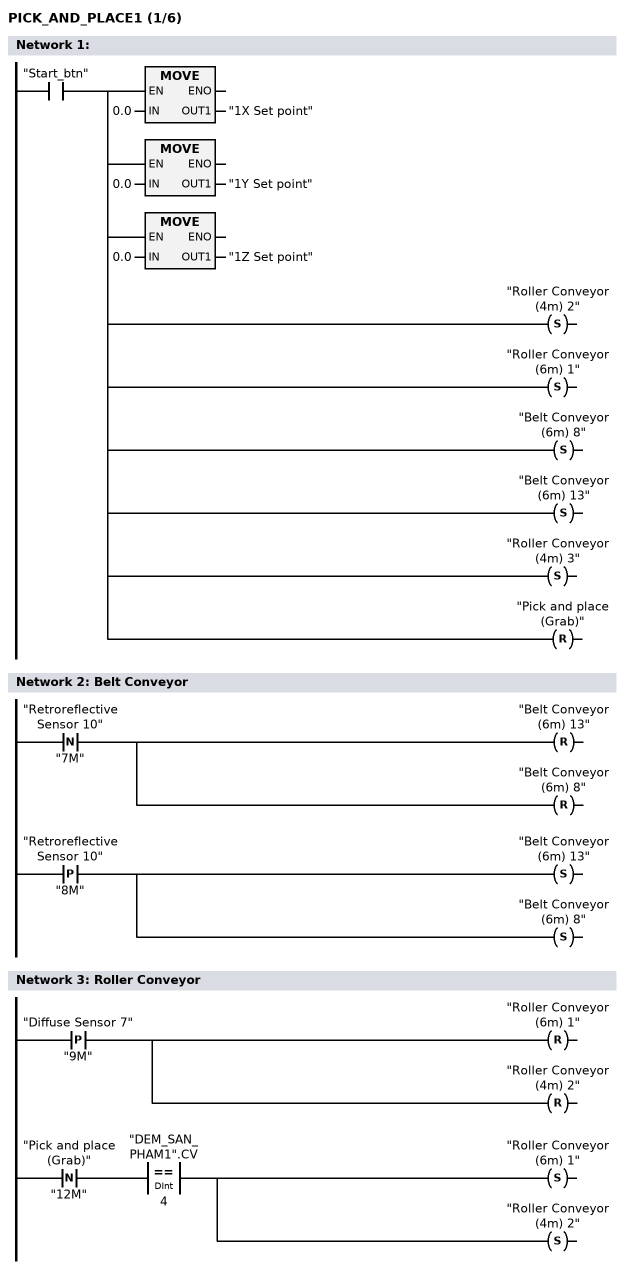
   RUNG wire#powerrail
      Contact( "Start_btn" )
      wire#w1
      Move(in := 0.0, out1 => "1X Set point")
   END_RUNG
   RUNG wire#w1
      Move(in := 0.0, out1 => "1Y Set point")
   END_RUNG
   RUNG wire#w1
      Move(in := 0.0, out1 => "1Z Set point")
   END_RUNG
   RUNG wire#w1
      S_Coil( "Roller Conveyor (4m) 2" )
   END_RUNG
   RUNG wire#w1
      S_Coil( "Roller Conveyor (6m) 1" )
   END_RUNG
   RUNG wire#w1
      S_Coil( "Belt Conveyor (6m) 8" )
   END_RUNG
   RUNG wire#w1
      S_Coil( "Belt Conveyor (6m) 13" )
   END_RUNG
   RUNG wire#w1
      S_Coil( "Roller Conveyor (4m) 3" )
   END_RUNG
   RUNG wire#w1
      R_Coil( "Pick and place (Grab)" )
   END_RUNG
   // the same network as SCL:
   IF "Start_btn" THEN
       "1X Set point" := 0.0;
       "1Y Set point" := 0.0;
       "1Z Set point" := 0.0;
       "Roller Conveyor (4m) 2" := TRUE;
       "Roller Conveyor (6m) 1" := TRUE;
       "Belt Conveyor (6m) 8" := TRUE;
       "Belt Conveyor (6m) 13" := TRUE;
       "Roller Conveyor (4m) 3" := TRUE;
       "Pick and place (Grab)" := FALSE;
   END_IF;
END_REGION

REGION Network 2: Belt Conveyor
   RUNG wire#powerrail
      N_Contact(operand := "Retroreflective Sensor 10", bit := "7M")
      wire#w1
      R_Coil( "Belt Conveyor (6m) 13" )
   END_RUNG
   RUNG wire#w1
      R_Coil( "Belt Conveyor (6m) 8" )
   END_RUNG
   RUNG wire#powerrail
      P_Contact(operand := "Retroreflective Sensor 10", bit := "8M")
      wire#w2
      S_Coil( "Belt Conveyor (6m) 13" )
   END_RUNG
   RUNG wire#w2
      S_Coil( "Belt Conveyor (6m) 8" )
   END_RUNG
   // the same network as SCL:
   #_w1 := NOT "Retroreflective Sensor 10" AND "7M";   // falling edge of "Retroreflective Sensor 10"
   "7M" := "Retroreflective Sensor 10";
   IF #_w1 THEN
       "Belt Conveyor (6m) 13" := FALSE;
       "Belt Conveyor (6m) 8" := FALSE;
   END_IF;
   #_w2 := "Retroreflective Sensor 10" AND NOT "8M";   // rising edge of "Retroreflective Sensor 10"
   "8M" := "Retroreflective Sensor 10";
   IF #_w2 THEN
       "Belt Conveyor (6m) 13" := TRUE;
       "Belt Conveyor (6m) 8" := TRUE;
   END_IF;
END_REGION

REGION Network 3: Roller Conveyor
   RUNG wire#powerrail
      P_Contact(operand := "Diffuse Sensor 7", bit := "9M")
      wire#w1
      R_Coil( "Roller Conveyor (6m) 1" )
   END_RUNG
   RUNG wire#w1
      R_Coil( "Roller Conveyor (4m) 2" )
   END_RUNG
   RUNG wire#powerrail
      N_Contact(operand := "Pick and place (Grab)", bit := "12M")
      { S7_Templates := "SrcType := DInt" } EQ_Contact(in1 := "DEM_SAN_PHAM1".CV, in2 := 4)
      wire#w2
      S_Coil( "Roller Conveyor (6m) 1" )
   END_RUNG
   RUNG wire#w2
      S_Coil( "Roller Conveyor (4m) 2" )
   END_RUNG
   // the same network as SCL:
   #_w1 := "Diffuse Sensor 7" AND NOT "9M";   // rising edge of "Diffuse Sensor 7"
   "9M" := "Diffuse Sensor 7";
   IF #_w1 THEN
       "Roller Conveyor (6m) 1" := FALSE;
       "Roller Conveyor (4m) 2" := FALSE;
   END_IF;
   #_w2 := NOT "Pick and place (Grab)" AND "12M";   // falling edge of "Pick and place (Grab)"
   "12M" := "Pick and place (Grab)";
   IF #_w2 AND ("DEM_SAN_PHAM1".CV = 4) THEN
       "Roller Conveyor (6m) 1" := TRUE;
       "Roller Conveyor (4m) 2" := TRUE;
   END_IF;
END_REGION

REGION Network 4
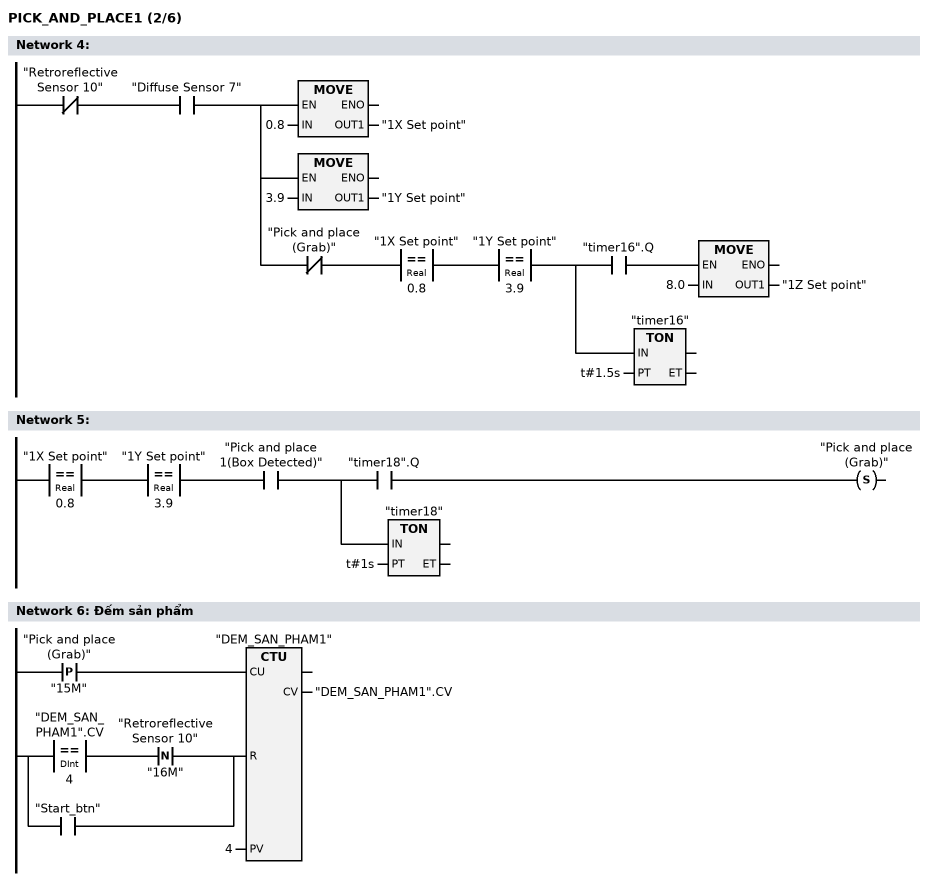
   #_w1 := NOT "Retroreflective Sensor 10" AND "Diffuse Sensor 7";
   IF #_w1 THEN
       "1X Set point" := 0.8;
       "1Y Set point" := 3.9;
   END_IF;
   #_w2 := #_w1 AND NOT "Pick and place (Grab)" AND ("1X Set point" = 0.8) AND ("1Y Set point" = 3.9);
   IF #_w2 AND "timer16".Q THEN "1Z Set point" := 8.0; END_IF;
   "timer16".TON(IN := #_w2, PT := t#1.5s);
END_REGION

REGION Network 5
   #_w1 := ("1X Set point" = 0.8) AND ("1Y Set point" = 3.9) AND "Pick and place 1(Box Detected)";
   IF #_w1 AND "timer18".Q THEN "Pick and place (Grab)" := TRUE; END_IF;
   "timer18".TON(IN := #_w1, PT := t#1s);
END_REGION

REGION Network 6: Đếm sản phẩm
   #_w1 := "Pick and place (Grab)" AND NOT "15M";   // rising edge of "Pick and place (Grab)"
   "15M" := "Pick and place (Grab)";
   #_w2 := ("DEM_SAN_PHAM1".CV = 4) AND NOT "Retroreflective Sensor 10" AND "16M";   // falling edge of "Retroreflective Sensor 10"
   "16M" := "Retroreflective Sensor 10";
   "DEM_SAN_PHAM1".CTU(CU := #_w1, R := #_w2 OR "Start_btn", PV := 4, CV => "DEM_SAN_PHAM1".CV);
END_REGION

REGION Network 7: SP 1
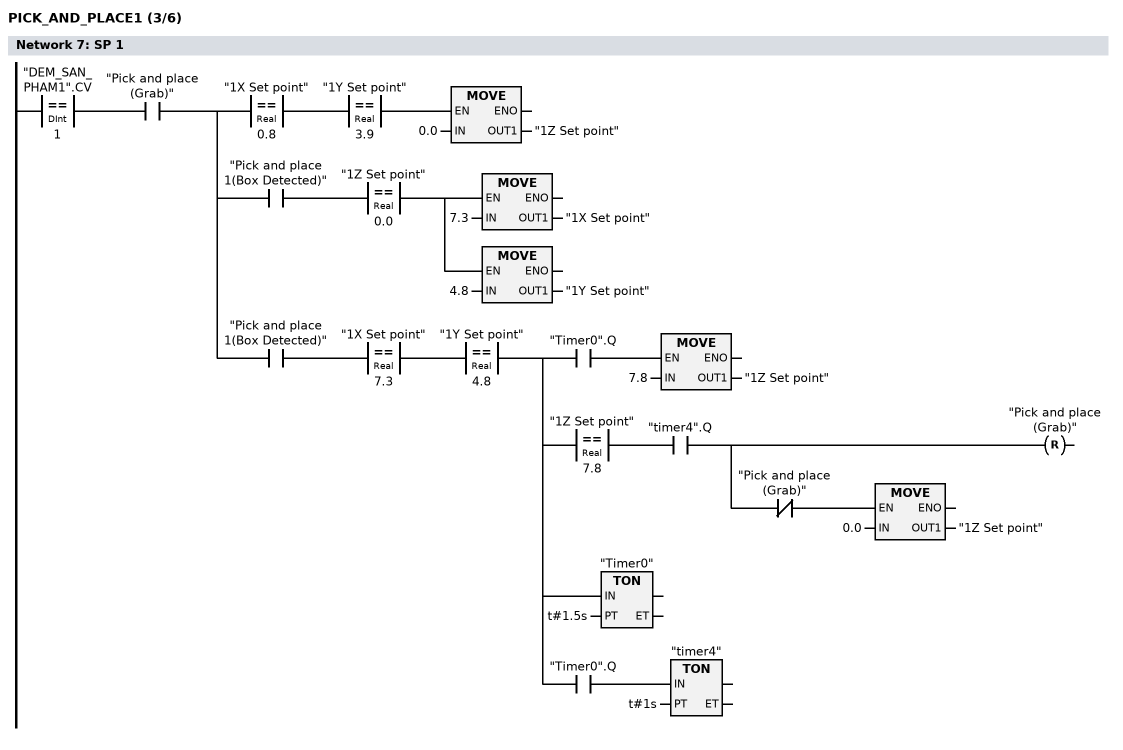
   #_w1 := ("DEM_SAN_PHAM1".CV = 1) AND "Pick and place (Grab)";
   IF #_w1 AND ("1X Set point" = 0.8) AND ("1Y Set point" = 3.9) THEN "1Z Set point" := 0.0; END_IF;
   IF #_w1 AND "Pick and place 1(Box Detected)" AND ("1Z Set point" = 0.0) THEN
       "1X Set point" := 7.3;
       "1Y Set point" := 4.8;
   END_IF;
   #_w2 := #_w1 AND "Pick and place 1(Box Detected)" AND ("1X Set point" = 7.3) AND ("1Y Set point" = 4.8);
   IF #_w2 AND "Timer0".Q THEN "1Z Set point" := 7.8; END_IF;
   #_w3 := #_w2 AND ("1Z Set point" = 7.8) AND "timer4".Q;
   IF #_w3 THEN "Pick and place (Grab)" := FALSE; END_IF;
   IF #_w3 AND NOT "Pick and place (Grab)" THEN "1Z Set point" := 0.0; END_IF;
   "Timer0".TON(IN := #_w2, PT := t#1.5s);
   "timer4".TON(IN := #_w2 AND "Timer0".Q, PT := t#1s);
END_REGION

REGION Network 8: SP 2
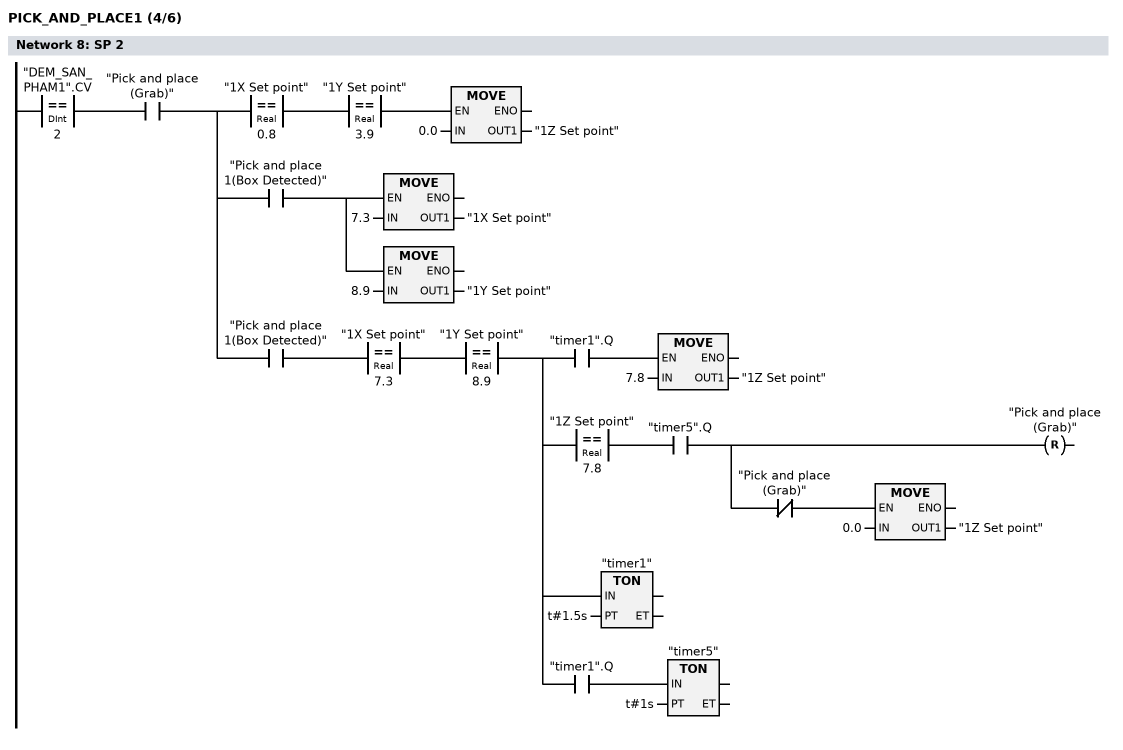
   #_w1 := ("DEM_SAN_PHAM1".CV = 2) AND "Pick and place (Grab)";
   IF #_w1 AND ("1X Set point" = 0.8) AND ("1Y Set point" = 3.9) THEN "1Z Set point" := 0.0; END_IF;
   IF #_w1 AND "Pick and place 1(Box Detected)" THEN
       "1X Set point" := 7.3;
       "1Y Set point" := 8.9;
   END_IF;
   #_w2 := #_w1 AND "Pick and place 1(Box Detected)" AND ("1X Set point" = 7.3) AND ("1Y Set point" = 8.9);
   IF #_w2 AND "timer1".Q THEN "1Z Set point" := 7.8; END_IF;
   #_w3 := #_w2 AND ("1Z Set point" = 7.8) AND "timer5".Q;
   IF #_w3 THEN "Pick and place (Grab)" := FALSE; END_IF;
   IF #_w3 AND NOT "Pick and place (Grab)" THEN "1Z Set point" := 0.0; END_IF;
   "timer1".TON(IN := #_w2, PT := t#1.5s);
   "timer5".TON(IN := #_w2 AND "timer1".Q, PT := t#1s);
END_REGION

REGION Network 9: SP 3
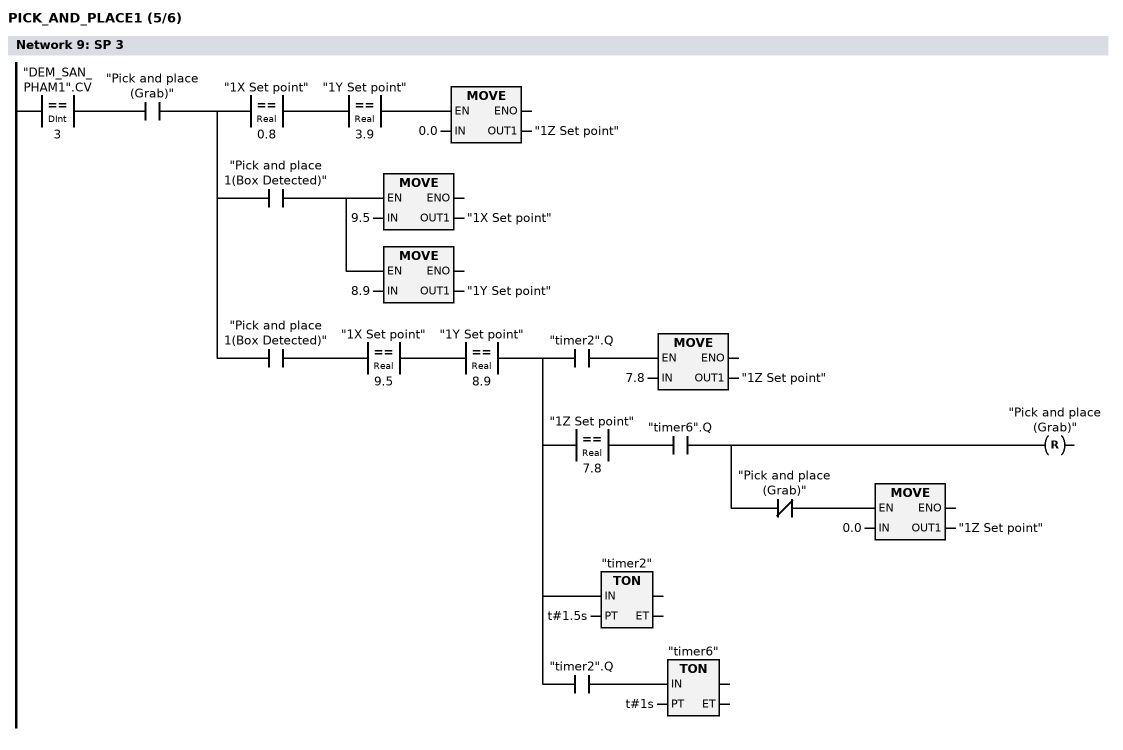
   #_w1 := ("DEM_SAN_PHAM1".CV = 3) AND "Pick and place (Grab)";
   IF #_w1 AND ("1X Set point" = 0.8) AND ("1Y Set point" = 3.9) THEN "1Z Set point" := 0.0; END_IF;
   IF #_w1 AND "Pick and place 1(Box Detected)" THEN
       "1X Set point" := 9.5;
       "1Y Set point" := 8.9;
   END_IF;
   #_w2 := #_w1 AND "Pick and place 1(Box Detected)" AND ("1X Set point" = 9.5) AND ("1Y Set point" = 8.9);
   IF #_w2 AND "timer2".Q THEN "1Z Set point" := 7.8; END_IF;
   #_w3 := #_w2 AND ("1Z Set point" = 7.8) AND "timer6".Q;
   IF #_w3 THEN "Pick and place (Grab)" := FALSE; END_IF;
   IF #_w3 AND NOT "Pick and place (Grab)" THEN "1Z Set point" := 0.0; END_IF;
   "timer2".TON(IN := #_w2, PT := t#1.5s);
   "timer6".TON(IN := #_w2 AND "timer2".Q, PT := t#1s);
END_REGION

REGION Network 10: SP 4
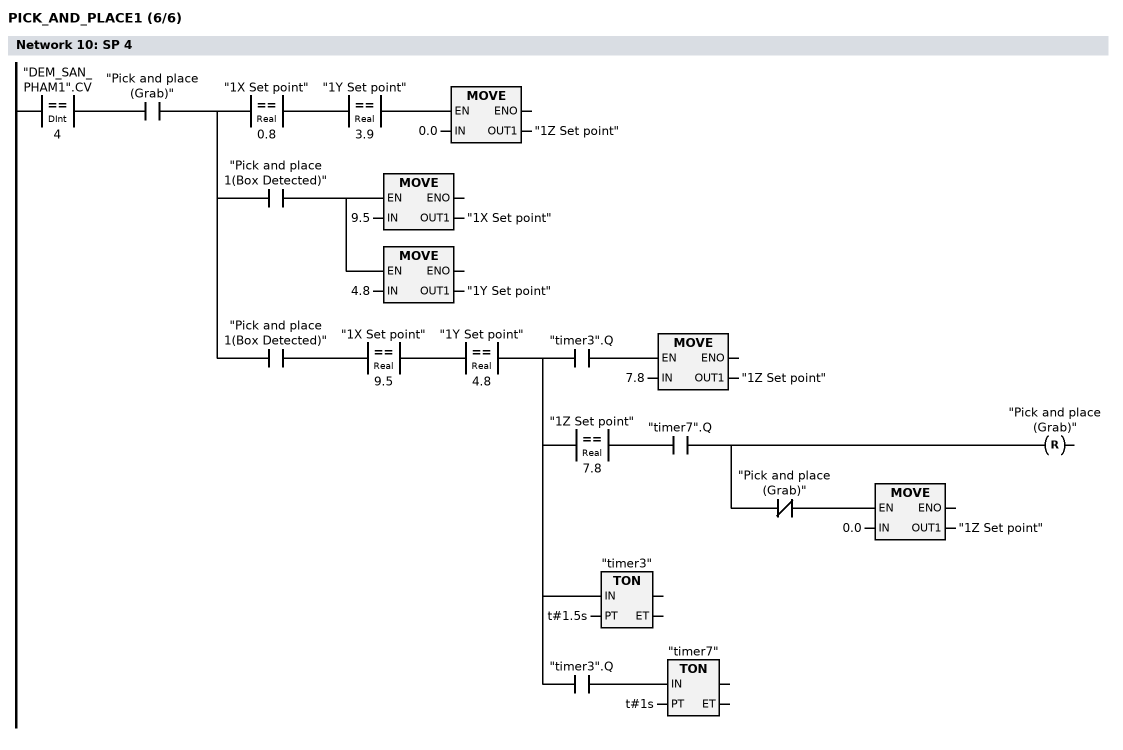
   #_w1 := ("DEM_SAN_PHAM1".CV = 4) AND "Pick and place (Grab)";
   IF #_w1 AND ("1X Set point" = 0.8) AND ("1Y Set point" = 3.9) THEN "1Z Set point" := 0.0; END_IF;
   IF #_w1 AND "Pick and place 1(Box Detected)" THEN
       "1X Set point" := 9.5;
       "1Y Set point" := 4.8;
   END_IF;
   #_w2 := #_w1 AND "Pick and place 1(Box Detected)" AND ("1X Set point" = 9.5) AND ("1Y Set point" = 4.8);
   IF #_w2 AND "timer3".Q THEN "1Z Set point" := 7.8; END_IF;
   #_w3 := #_w2 AND ("1Z Set point" = 7.8) AND "timer7".Q;
   IF #_w3 THEN "Pick and place (Grab)" := FALSE; END_IF;
   IF #_w3 AND NOT "Pick and place (Grab)" THEN "1Z Set point" := 0.0; END_IF;
   "timer3".TON(IN := #_w2, PT := t#1.5s);
   "timer7".TON(IN := #_w2 AND "timer3".Q, PT := t#1s);
END_REGION
END_FUNCTION

FUNCTION "PICK_AND_PLACE2" : Void   // FC6, LAD
{ S7_Optimized_Access := 'TRUE' }
VERSION : 0.1
   VAR_TEMP   // added for the SCL form of the ladder/FBD networks
      _w1 : Bool;
      _w2 : Bool;
      _w3 : Bool;
   END_VAR
BEGIN

REGION Network 1
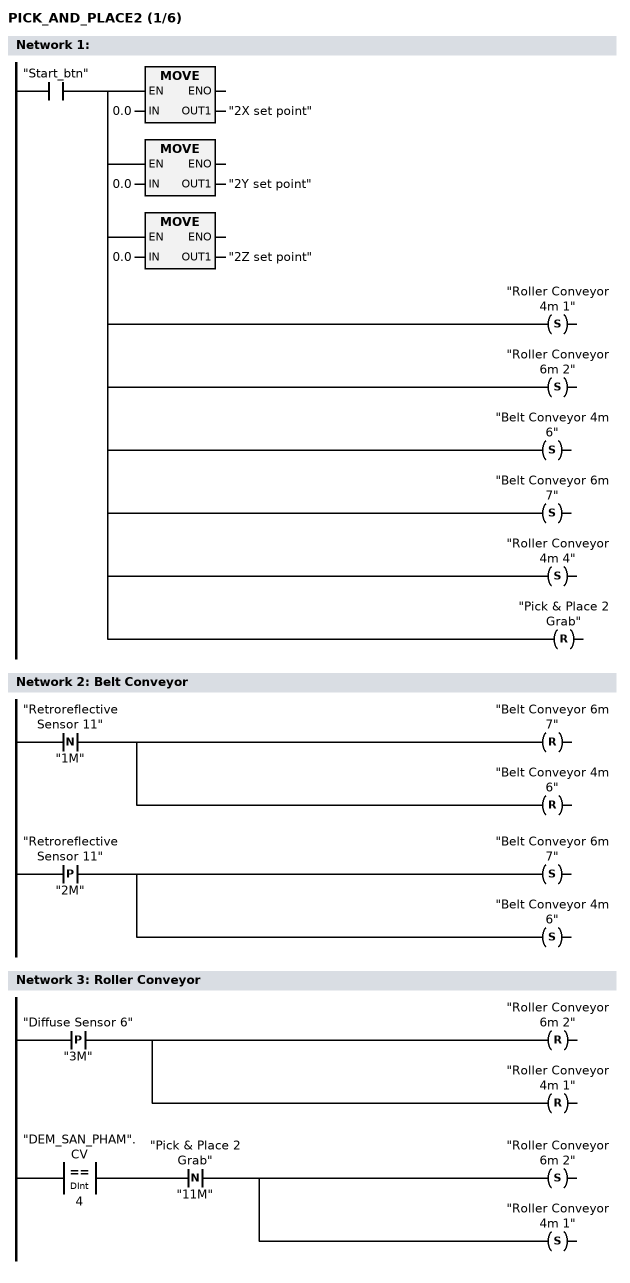
   RUNG wire#powerrail
      Contact( "Start_btn" )
      wire#w1
      Move(in := 0.0, out1 => "2X set point")
   END_RUNG
   RUNG wire#w1
      Move(in := 0.0, out1 => "2Y set point")
   END_RUNG
   RUNG wire#w1
      Move(in := 0.0, out1 => "2Z set point")
   END_RUNG
   RUNG wire#w1
      S_Coil( "Roller Conveyor 4m 1" )
   END_RUNG
   RUNG wire#w1
      S_Coil( "Roller Conveyor 6m 2" )
   END_RUNG
   RUNG wire#w1
      S_Coil( "Belt Conveyor 4m 6" )
   END_RUNG
   RUNG wire#w1
      S_Coil( "Belt Conveyor 6m 7" )
   END_RUNG
   RUNG wire#w1
      S_Coil( "Roller Conveyor 4m 4" )
   END_RUNG
   RUNG wire#w1
      R_Coil( "Pick & Place 2 Grab" )
   END_RUNG
   // the same network as SCL:
   IF "Start_btn" THEN
       "2X set point" := 0.0;
       "2Y set point" := 0.0;
       "2Z set point" := 0.0;
       "Roller Conveyor 4m 1" := TRUE;
       "Roller Conveyor 6m 2" := TRUE;
       "Belt Conveyor 4m 6" := TRUE;
       "Belt Conveyor 6m 7" := TRUE;
       "Roller Conveyor 4m 4" := TRUE;
       "Pick & Place 2 Grab" := FALSE;
   END_IF;
END_REGION

REGION Network 2: Belt Conveyor
   RUNG wire#powerrail
      N_Contact(operand := "Retroreflective Sensor 11", bit := "1M")
      wire#w1
      R_Coil( "Belt Conveyor 6m 7" )
   END_RUNG
   RUNG wire#w1
      R_Coil( "Belt Conveyor 4m 6" )
   END_RUNG
   RUNG wire#powerrail
      P_Contact(operand := "Retroreflective Sensor 11", bit := "2M")
      wire#w2
      S_Coil( "Belt Conveyor 6m 7" )
   END_RUNG
   RUNG wire#w2
      S_Coil( "Belt Conveyor 4m 6" )
   END_RUNG
   // the same network as SCL:
   #_w1 := NOT "Retroreflective Sensor 11" AND "1M";   // falling edge of "Retroreflective Sensor 11"
   "1M" := "Retroreflective Sensor 11";
   IF #_w1 THEN
       "Belt Conveyor 6m 7" := FALSE;
       "Belt Conveyor 4m 6" := FALSE;
   END_IF;
   #_w2 := "Retroreflective Sensor 11" AND NOT "2M";   // rising edge of "Retroreflective Sensor 11"
   "2M" := "Retroreflective Sensor 11";
   IF #_w2 THEN
       "Belt Conveyor 6m 7" := TRUE;
       "Belt Conveyor 4m 6" := TRUE;
   END_IF;
END_REGION

REGION Network 3: Roller Conveyor
   RUNG wire#powerrail
      P_Contact(operand := "Diffuse Sensor 6", bit := "3M")
      wire#w1
      R_Coil( "Roller Conveyor 6m 2" )
   END_RUNG
   RUNG wire#w1
      R_Coil( "Roller Conveyor 4m 1" )
   END_RUNG
   RUNG wire#powerrail
      { S7_Templates := "SrcType := DInt" } EQ_Contact(in1 := "DEM_SAN_PHAM".CV, in2 := 4)
      N_Contact(operand := "Pick & Place 2 Grab", bit := "11M")
      wire#w2
      S_Coil( "Roller Conveyor 6m 2" )
   END_RUNG
   RUNG wire#w2
      S_Coil( "Roller Conveyor 4m 1" )
   END_RUNG
   // the same network as SCL:
   #_w1 := "Diffuse Sensor 6" AND NOT "3M";   // rising edge of "Diffuse Sensor 6"
   "3M" := "Diffuse Sensor 6";
   IF #_w1 THEN
       "Roller Conveyor 6m 2" := FALSE;
       "Roller Conveyor 4m 1" := FALSE;
   END_IF;
   #_w2 := ("DEM_SAN_PHAM".CV = 4) AND NOT "Pick & Place 2 Grab" AND "11M";   // falling edge of "Pick & Place 2 Grab"
   "11M" := "Pick & Place 2 Grab";
   IF #_w2 THEN
       "Roller Conveyor 6m 2" := TRUE;
       "Roller Conveyor 4m 1" := TRUE;
   END_IF;
END_REGION

REGION Network 4
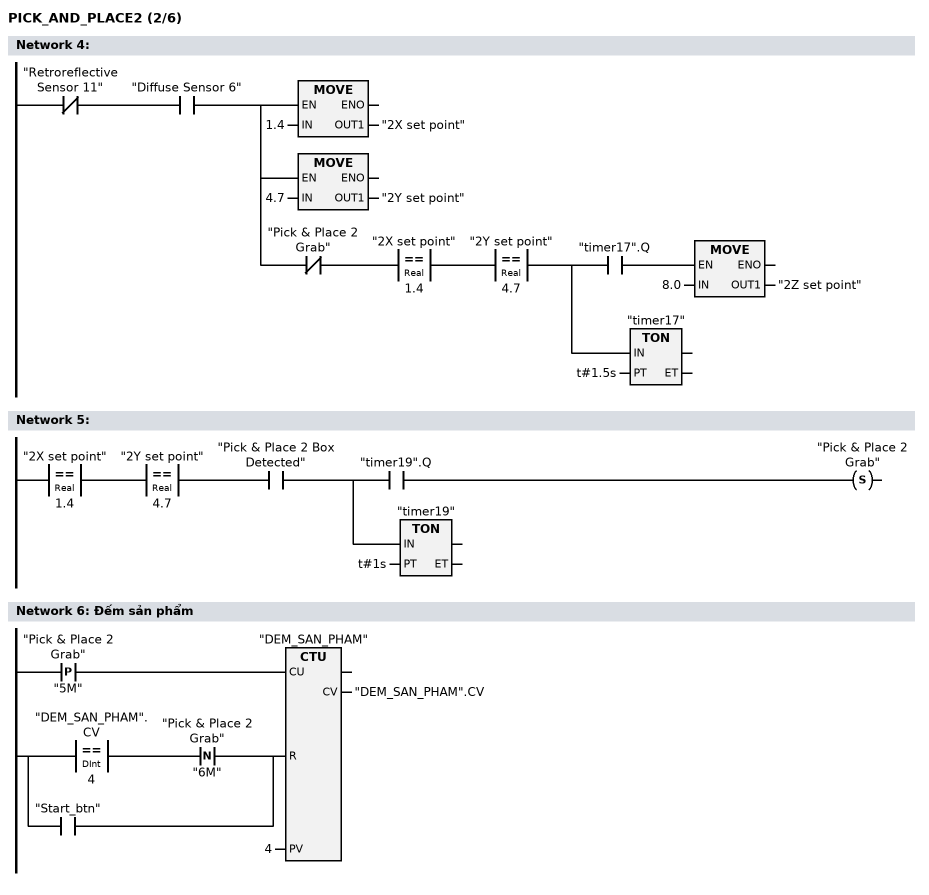
   #_w1 := NOT "Retroreflective Sensor 11" AND "Diffuse Sensor 6";
   IF #_w1 THEN
       "2X set point" := 1.4;
       "2Y set point" := 4.7;
   END_IF;
   #_w2 := #_w1 AND NOT "Pick & Place 2 Grab" AND ("2X set point" = 1.4) AND ("2Y set point" = 4.7);
   IF #_w2 AND "timer17".Q THEN "2Z set point" := 8.0; END_IF;
   "timer17".TON(IN := #_w2, PT := t#1.5s);
END_REGION

REGION Network 5
   #_w1 := ("2X set point" = 1.4) AND ("2Y set point" = 4.7) AND "Pick & Place 2 Box Detected";
   IF #_w1 AND "timer19".Q THEN "Pick & Place 2 Grab" := TRUE; END_IF;
   "timer19".TON(IN := #_w1, PT := t#1s);
END_REGION

REGION Network 6: Đếm sản phẩm
   #_w1 := "Pick & Place 2 Grab" AND NOT "5M";   // rising edge of "Pick & Place 2 Grab"
   "5M" := "Pick & Place 2 Grab";
   #_w2 := ("DEM_SAN_PHAM".CV = 4) AND NOT "Pick & Place 2 Grab" AND "6M";   // falling edge of "Pick & Place 2 Grab"
   "6M" := "Pick & Place 2 Grab";
   "DEM_SAN_PHAM".CTU(CU := #_w1, R := #_w2 OR "Start_btn", PV := 4, CV => "DEM_SAN_PHAM".CV);
END_REGION

REGION Network 7: SP 1
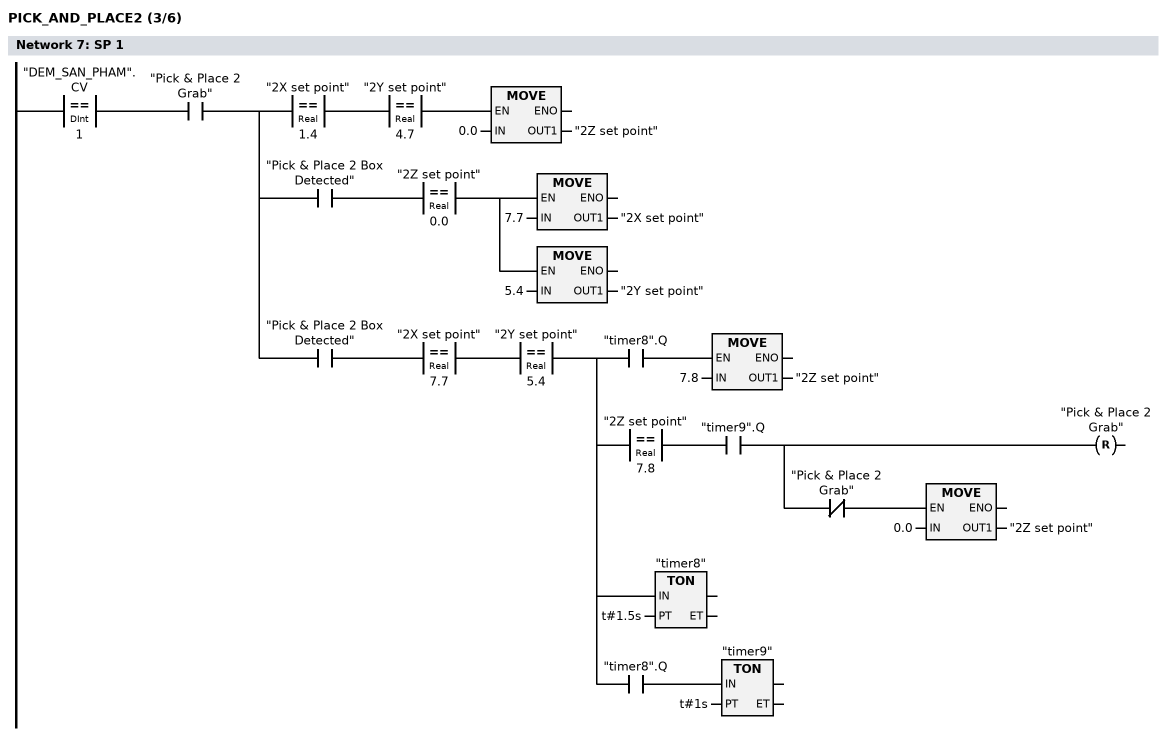
   #_w1 := ("DEM_SAN_PHAM".CV = 1) AND "Pick & Place 2 Grab";
   IF #_w1 AND ("2X set point" = 1.4) AND ("2Y set point" = 4.7) THEN "2Z set point" := 0.0; END_IF;
   IF #_w1 AND "Pick & Place 2 Box Detected" AND ("2Z set point" = 0.0) THEN
       "2X set point" := 7.7;
       "2Y set point" := 5.4;
   END_IF;
   #_w2 := #_w1 AND "Pick & Place 2 Box Detected" AND ("2X set point" = 7.7) AND ("2Y set point" = 5.4);
   IF #_w2 AND "timer8".Q THEN "2Z set point" := 7.8; END_IF;
   #_w3 := #_w2 AND ("2Z set point" = 7.8) AND "timer9".Q;
   IF #_w3 THEN "Pick & Place 2 Grab" := FALSE; END_IF;
   IF #_w3 AND NOT "Pick & Place 2 Grab" THEN "2Z set point" := 0.0; END_IF;
   "timer8".TON(IN := #_w2, PT := t#1.5s);
   "timer9".TON(IN := #_w2 AND "timer8".Q, PT := t#1s);
END_REGION

REGION Network 8: SP 2
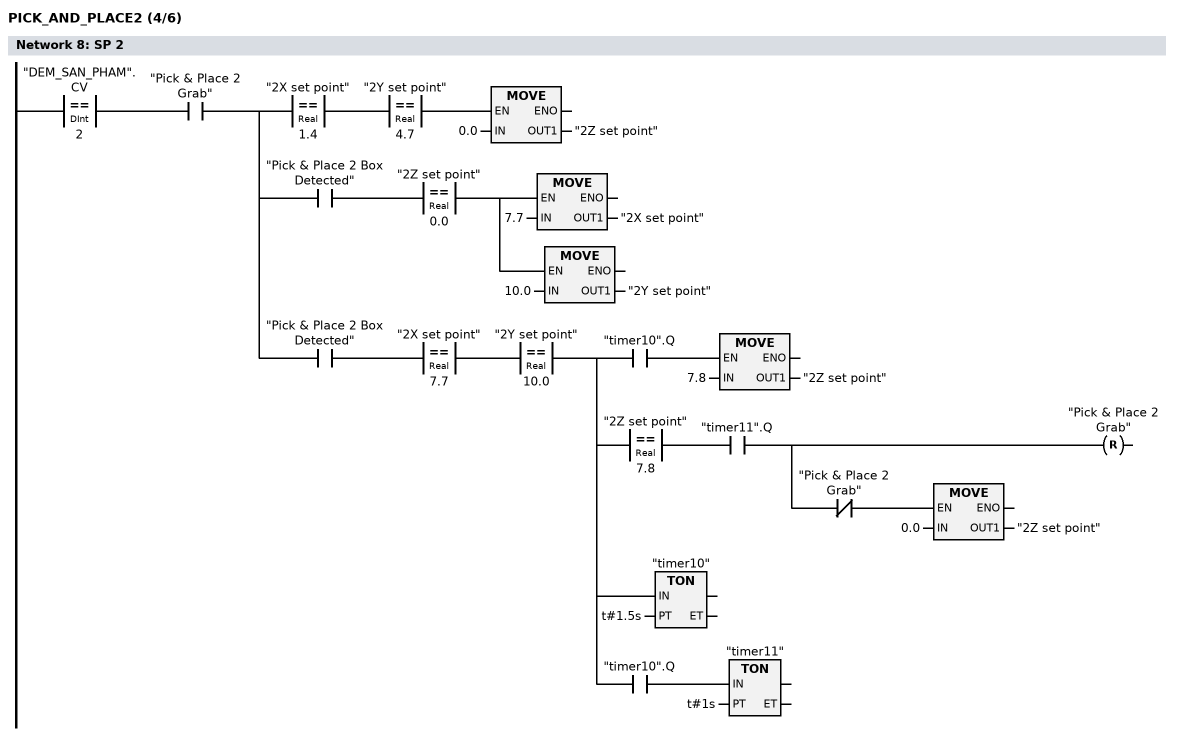
   #_w1 := ("DEM_SAN_PHAM".CV = 2) AND "Pick & Place 2 Grab";
   IF #_w1 AND ("2X set point" = 1.4) AND ("2Y set point" = 4.7) THEN "2Z set point" := 0.0; END_IF;
   IF #_w1 AND "Pick & Place 2 Box Detected" AND ("2Z set point" = 0.0) THEN
       "2X set point" := 7.7;
       "2Y set point" := 10.0;
   END_IF;
   #_w2 := #_w1 AND "Pick & Place 2 Box Detected" AND ("2X set point" = 7.7) AND ("2Y set point" = 10.0);
   IF #_w2 AND "timer10".Q THEN "2Z set point" := 7.8; END_IF;
   #_w3 := #_w2 AND ("2Z set point" = 7.8) AND "timer11".Q;
   IF #_w3 THEN "Pick & Place 2 Grab" := FALSE; END_IF;
   IF #_w3 AND NOT "Pick & Place 2 Grab" THEN "2Z set point" := 0.0; END_IF;
   "timer10".TON(IN := #_w2, PT := t#1.5s);
   "timer11".TON(IN := #_w2 AND "timer10".Q, PT := t#1s);
END_REGION

REGION Network 9: SP 3
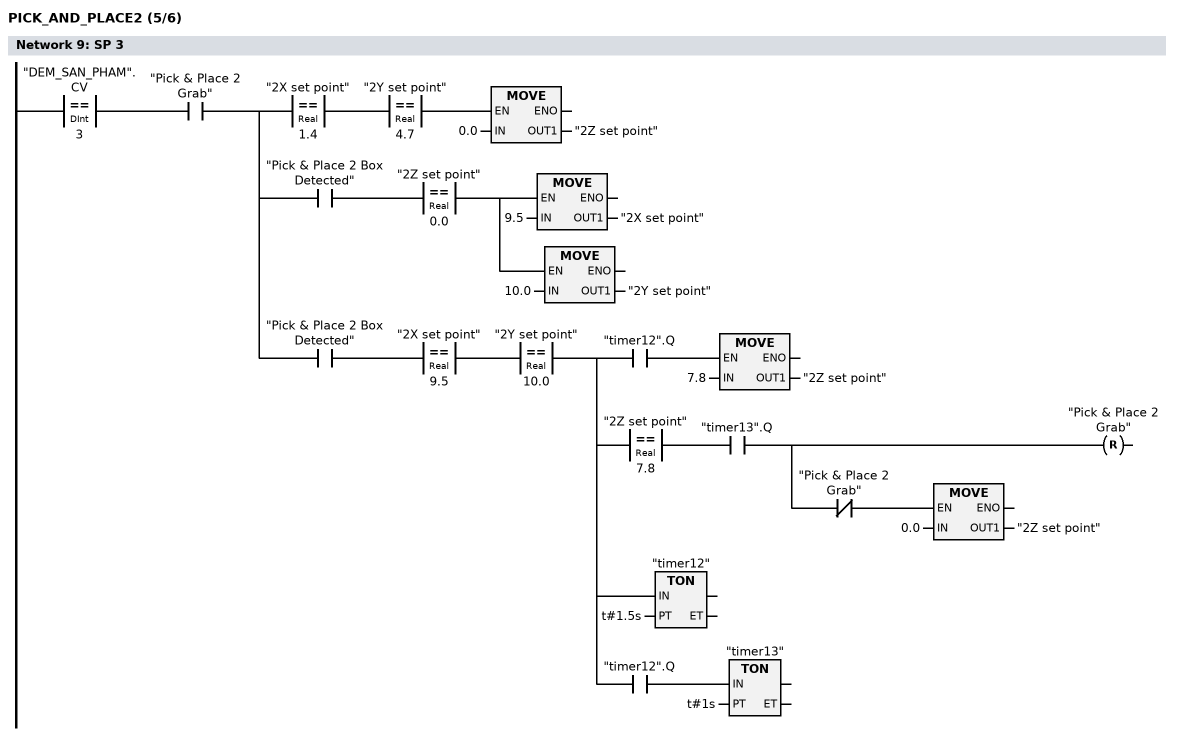
   #_w1 := ("DEM_SAN_PHAM".CV = 3) AND "Pick & Place 2 Grab";
   IF #_w1 AND ("2X set point" = 1.4) AND ("2Y set point" = 4.7) THEN "2Z set point" := 0.0; END_IF;
   IF #_w1 AND "Pick & Place 2 Box Detected" AND ("2Z set point" = 0.0) THEN
       "2X set point" := 9.5;
       "2Y set point" := 10.0;
   END_IF;
   #_w2 := #_w1 AND "Pick & Place 2 Box Detected" AND ("2X set point" = 9.5) AND ("2Y set point" = 10.0);
   IF #_w2 AND "timer12".Q THEN "2Z set point" := 7.8; END_IF;
   #_w3 := #_w2 AND ("2Z set point" = 7.8) AND "timer13".Q;
   IF #_w3 THEN "Pick & Place 2 Grab" := FALSE; END_IF;
   IF #_w3 AND NOT "Pick & Place 2 Grab" THEN "2Z set point" := 0.0; END_IF;
   "timer12".TON(IN := #_w2, PT := t#1.5s);
   "timer13".TON(IN := #_w2 AND "timer12".Q, PT := t#1s);
END_REGION

REGION Network 10: SP 4
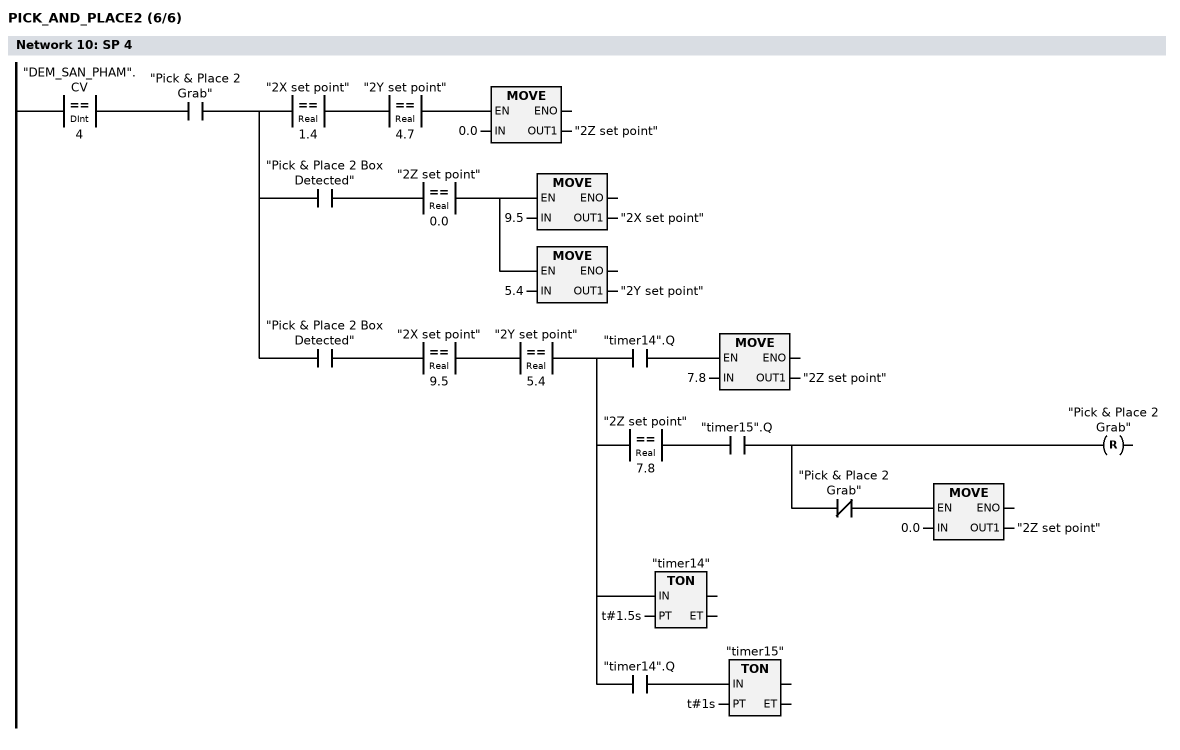
   #_w1 := ("DEM_SAN_PHAM".CV = 4) AND "Pick & Place 2 Grab";
   IF #_w1 AND ("2X set point" = 1.4) AND ("2Y set point" = 4.7) THEN "2Z set point" := 0.0; END_IF;
   IF #_w1 AND "Pick & Place 2 Box Detected" AND ("2Z set point" = 0.0) THEN
       "2X set point" := 9.5;
       "2Y set point" := 5.4;
   END_IF;
   #_w2 := #_w1 AND "Pick & Place 2 Box Detected" AND ("2X set point" = 9.5) AND ("2Y set point" = 5.4);
   IF #_w2 AND "timer14".Q THEN "2Z set point" := 7.8; END_IF;
   #_w3 := #_w2 AND ("2Z set point" = 7.8) AND "timer15".Q;
   IF #_w3 THEN "Pick & Place 2 Grab" := FALSE; END_IF;
   IF #_w3 AND NOT "Pick & Place 2 Grab" THEN "2Z set point" := 0.0; END_IF;
   "timer14".TON(IN := #_w2, PT := t#1.5s);
   "timer15".TON(IN := #_w2 AND "timer14".Q, PT := t#1s);
END_REGION
END_FUNCTION

FUNCTION "MHJ-PLC-Lab-Function-S71200" : Void   // FC9000, SCL
{ S7_Optimized_Access := 'TRUE' }
VERSION : 0.1
   VAR_TEMP
      rdTimeReturn : Int;
      outputTime : DTL;
      SyncVal : Byte;
      forVal : Int;
      forVal_2 : Int;
      Value : Byte;
   END_VAR
   VAR CONSTANT
      CompVal : Byte := 16#34;
      Value_01 : Byte := 16#11;
      Value_01_DW : DWord := 16#A165_D992;
      Value_02_DW : DWord := 16#58BE_4401;
   END_VAR
BEGIN

   #Value:=PEEK(area := 16#82,
        dbNumber := 0,
        byteOffset := 511);
   #Value := #Value + 1;

   POKE(area := 16#82,
        dbNumber := 0,
        byteOffset := 511,
        value := #Value);

   POKE(area:=16#81,
        dbNumber:=0,
        byteOffset:=1016,
        value:=#Value_01_DW);
   POKE(area := 16#81,
        dbNumber := 0,
        byteOffset := 1020,
        value := #Value_02_DW);

   POKE(area := 16#81,
        dbNumber := 0,
        byteOffset := 511,
        value := B#16#00);

   FOR #forVal := 0 TO 120 DO
       FOR #forVal_2:=0 TO 10 DO
           #rdTimeReturn:=RD_SYS_T(#outputTime);
           #rdTimeReturn := WR_SYS_T(#outputTime);
           #rdTimeReturn := RD_SYS_T(#outputTime);
           #rdTimeReturn := WR_SYS_T(#outputTime);
       END_FOR;
       #SyncVal:= PEEK(area := 16#81,
                      dbNumber := 0,
                      byteOffset := 511);
       IF #SyncVal = #CompVal THEN
          GOTO M_1;
       END_IF;
   END_FOR;
   RETURN;

   M_1:
   POKE(area := 16#81,
        dbNumber := 0,
        byteOffset := 511,
        value := B#16#0);
END_FUNCTION

ORGANIZATION_BLOCK "Main_1"   // OB123, LAD, ProgramCycle
TITLE = "Main Program Sweep (Cycle)"
{ S7_Optimized_Access := 'TRUE' }
VERSION : 0.1
   VAR_INPUT
      Initial_Call : Bool;   // Initial call of this OB
      Remanence : Bool;   // =True, if remanent data are available
   END_VAR
BEGIN

REGION Network 1
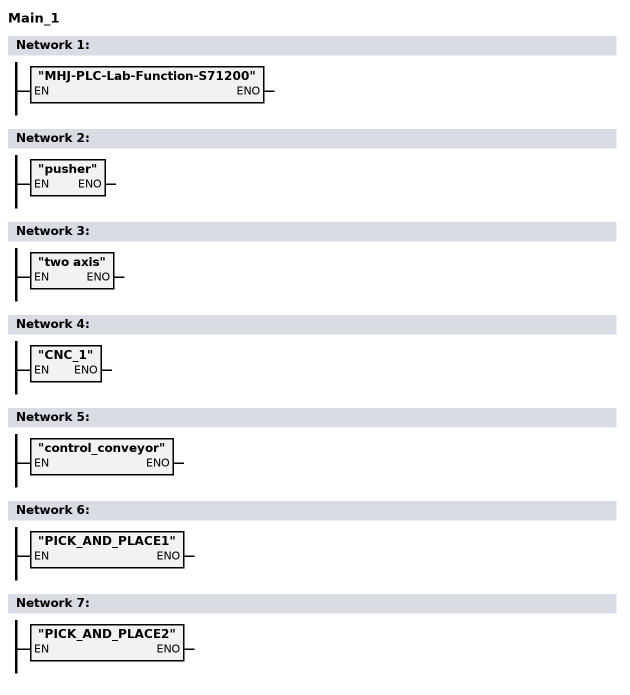
   RUNG wire#powerrail
      "MHJ-PLC-Lab-Function-S71200"()
   END_RUNG
   // the same network as SCL:
   "MHJ-PLC-Lab-Function-S71200"();
END_REGION

REGION Network 2
   RUNG wire#powerrail
      "pusher"()
   END_RUNG
   // the same network as SCL:
   "pusher"();
END_REGION

REGION Network 3
   RUNG wire#powerrail
      "two axis"()
   END_RUNG
   // the same network as SCL:
   "two axis"();
END_REGION

REGION Network 4
   RUNG wire#powerrail
      "CNC_1"()
   END_RUNG
   // the same network as SCL:
   "CNC_1"();
END_REGION

REGION Network 5
   RUNG wire#powerrail
      "control_conveyor"()
   END_RUNG
   // the same network as SCL:
   "control_conveyor"();
END_REGION

REGION Network 6
   RUNG wire#powerrail
      "PICK_AND_PLACE1"()
   END_RUNG
   // the same network as SCL:
   "PICK_AND_PLACE1"();
END_REGION

REGION Network 7
   RUNG wire#powerrail
      "PICK_AND_PLACE2"()
   END_RUNG
   // the same network as SCL:
   "PICK_AND_PLACE2"();
END_REGION
END_ORGANIZATION_BLOCK